# B&R Automation Studio project Hybrid
Automation Studio 6.3.4.31; Oval trak demo with one conveyor segment; technology packages: mappCockpit 6.2.1, mappMotion 6.7.0, mappServices 6.2.0, mappView 6.2.0, OpcUaCs 6.0.0

## Configuration APC2200

CPU 5APC2200.AL14-000, AutomationRuntime 6.3.4, Build 11.3.0, Vc 6.0.0

### Task classes (Cpu.sw)
```
Cyclic#1 (cycle 800 us, tolerance 0 us):
  Main <- Main.prg
DataObjects: McAcpSys
NcDataObjects: McDriveLog
Binaries: FWRules, McAcpSim, ArSvcReg, TCData, McAcpDrv, udbdef, iomap, Config_1, BRRole, arconfig, asfw, Config_5, ashwac, sysconf, User, Config_4, Role, UaCsConfig, ashwd, Config_3, Config_2
Libraries: astime, UaCoal, powerlnk, sys_lib, UaCoalPrv, AsIODiag, runtime, AsBrStr, CoTrace, AsZip, FileIO, MpBase, standard, McBase, McAcpAx, McAxis, MpAxis, McPureVAx, McAcpTrak
```

### Hardware
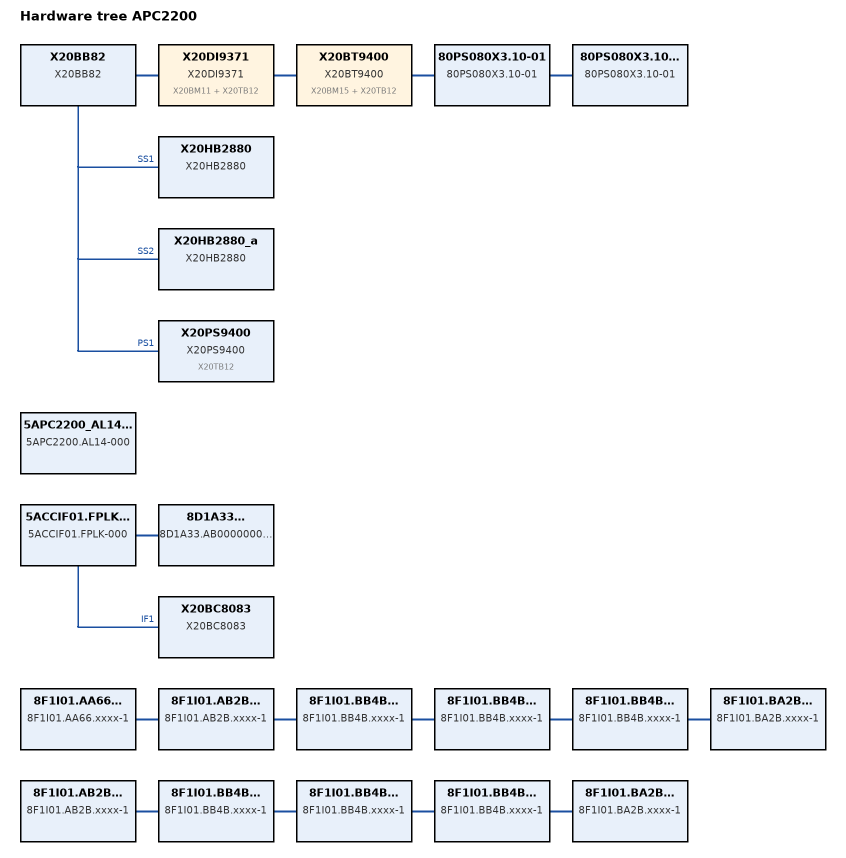
```
5ACCIF01.FPLK-000 : 5ACCIF01.FPLK-000 v1.9.0.0  [PLK2 -> 8D1A33.AB0000000-1.PLK1 [Cable Type=PowerlinkCable, Length=10, Version=1.0.0.3]; SL -> 5APC2200_AL14_000.SL1]
  Connector IF1:
    CycleTime = 800
    EplNatSubnet = 192.168.102.0
    Channel1
    ChannelID1 = McAcpBroadcast
    ChannelType1 = OCTET[120]
5APC2200_AL14_000 : 5APC2200.AL14-000 v2.0.7.0
  Connector IF3:
    AssignedOperatingSystem = ARemb
    ActivateDevice = 1
    HostName = llm-demosystem-ds3
    Mode = Manual
    InternetAddress = 10.43.39.206
    SubnetMask = 255.255.255.0
    InaNodeNumber = 206
    ActivateSnmp = 2
  Connector IF4:
    AssignedOperatingSystem = ARemb
    ActivateDevice = 1
    HostName = llm-demosystem-ds3
    ActivateSnmp = 2
  Connector IF5:
    AssignedOperatingSystem = ARemb
  Connector IF6:
    AssignedOperatingSystem = ARemb
  ConfigurationID = Hybrid_APC910
  Simulation = 1
  MotionLoggerSize = 2048000
  TimerDeviceType = EPLX2X
  TimerDevice = 5ACCIF01.FPLK-000.IF1
  TaskClassIdleTime = 1600
  Cyclic1Duration = 800
  Cyclic1Tolerance = 0
  Cyclic3Duration = 49600
  Cyclic3Tolerance = 49600
  Cyclic8Duration = 9600
  FileDevice1
  FileDeviceName1 = SvgData
  FileDevicePath1 = USER_PATH
  EthernetHostName = llm-demosystem-ds3
  EthernetDefaultGateway = 10.43.39.1
  ActivateFtpServer = 1
  FTPProtocol = 1
  FtpUser1
  FtpUsername1 = Admin
  FtpUserPassword1 = Pdt4iUtP2akYp0fWOPx8iCFOek96otsGjJ7w2jsAU3U=
  FtpUserSalt1 = ubly4TPI
  FTPAccessRight1 = 0
  ActivateWebServer = 1
  WebServerProtocol = 3
  ActivateSdm = 1
80PS080X3.10-01 : 80PS080X3.10-01 v1.7.0.0  [X2X1 -> X20BT9400.X2X1 [Cable Type=X2XCable, Length=10, Version=1.0.0.3]]
  Supervision = off
  ParallelMode01 = on
  VoltageSet01 = 58
  RampMode01 = steep
  ChopperEnable01 = on
80PS080X3.10-01_a : 80PS080X3.10-01 v1.7.0.0  [X2X1 -> 80PS080X3.10-01.X2X2 [Cable Type=X2XCable, Length=10, Version=1.0.0.3]]
  Supervision = off
  ParallelMode01 = on
  VoltageSet01 = 58
  RampMode01 = steep
  ChopperEnable01 = on
8D1A33.AB0000000-1 : 8D1A33.AB0000000-1 v1.0.1.0 (NodeNumber=130)  [PLK1 -> 5ACCIF01.FPLK-000.PLK2 [Cable Type=PowerlinkCable, Length=10, Version=1.0.0.3]]
  DriveConfiguration/Channel[1]/RealAxis:
    AxisReference = gAxis_1
  DriveConfiguration/Channel[1]/RealAxis/MechanicalElements/RotaryToLinearTransformation:
    ReferenceDistance = 0.13
8F1I01.AA66.Seg_0 : 8F1I01.AA66.xxxx-1 v1.0.0.4 (NodeNumber=7)  [PLK1 -> 8F1I01.BA2B.xxxx-1_a.PLK2 [Cable Type=PowerlinkCable, Length=10, Version=1.0.0.3]; PLK2 -> 8F1I01.AB2B.xxxx-1.PLK1 [Cable Type=PowerlinkCable, Length=10, Version=1.0.0.3]; PLK3 -> X20BC8083.PLK2 [Cable Type=PowerlinkCable, Length=10, Version=1.0.0.3]]
  EnableDNA = on
  DriveConfiguration/Segment:
    SegmentReference = Seg_01
8F1I01.AB2B.xxxx-1 : 8F1I01.AB2B.xxxx-1 v1.0.0.4 (NodeNumber=8)  [PLK1 -> 8F1I01.AA66.Seg_0.PLK2 [Cable Type=PowerlinkCable, Length=10, Version=1.0.0.3]; PLK2 -> 8F1I01.BB4B.xxxx-1.PLK1 [Cable Type=PowerlinkCable, Length=10, Version=1.0.0.3]]
  EnableDNA = on
  DriveConfiguration/Segment:
    SegmentReference = Seg_02
8F1I01.AB2B.xxxx-1_a : 8F1I01.AB2B.xxxx-1 v1.0.0.4 (NodeNumber=2)  [PLK2 -> 8F1I01.BB4B.xxxx-1_e.PLK1 [Cable Type=PowerlinkCable, Length=10, Version=1.0.0.3]]
  EnableDNA = on
  DriveConfiguration/Segment:
    SegmentReference = Seg_08
    SegmentSectorReference = SegSec_08
8F1I01.BA2B.xxxx-1 : 8F1I01.BA2B.xxxx-1 v1.0.0.4 (NodeNumber=12)  [PLK1 -> 8F1I01.BB4B.xxxx-1_b.PLK2 [Cable Type=PowerlinkCable, Length=10, Version=1.0.0.3]]
  EnableDNA = on
  DriveConfiguration/Segment:
    SegmentReference = Seg_06
    SegmentSectorReference = SegSec_06
8F1I01.BA2B.xxxx-1_a : 8F1I01.BA2B.xxxx-1 v1.0.0.4 (NodeNumber=6)  [PLK1 -> 8F1I01.BB4B.xxxx-1_c.PLK2 [Cable Type=PowerlinkCable, Length=10, Version=1.0.0.3]; PLK2 -> 8F1I01.AA66.Seg_0.PLK1 [Cable Type=PowerlinkCable, Length=10, Version=1.0.0.3]]
  EnableDNA = on
  DriveConfiguration/Segment:
    SegmentReference = Seg_12
8F1I01.BB4B.xxxx-1 : 8F1I01.BB4B.xxxx-1 v1.0.0.4 (NodeNumber=9)  [PLK1 -> 8F1I01.AB2B.xxxx-1.PLK2 [Cable Type=PowerlinkCable, Length=10, Version=1.0.0.3]; PLK2 -> 8F1I01.BB4B.xxxx-1_a.PLK1 [Cable Type=PowerlinkCable, Length=10, Version=1.0.0.3]]
  EnableDNA = on
  DriveConfiguration/Segment:
    SegmentReference = Seg_03
8F1I01.BB4B.xxxx-1_a : 8F1I01.BB4B.xxxx-1 v1.0.0.4 (NodeNumber=10)  [PLK1 -> 8F1I01.BB4B.xxxx-1.PLK2 [Cable Type=PowerlinkCable, Length=10, Version=1.0.0.3]; PLK2 -> 8F1I01.BB4B.xxxx-1_b.PLK1 [Cable Type=PowerlinkCable, Length=10, Version=1.0.0.3]]
  EnableDNA = on
  DriveConfiguration/Segment:
    SegmentReference = Seg_04
8F1I01.BB4B.xxxx-1_b : 8F1I01.BB4B.xxxx-1 v1.0.0.4 (NodeNumber=11)  [PLK1 -> 8F1I01.BB4B.xxxx-1_a.PLK2 [Cable Type=PowerlinkCable, Length=10, Version=1.0.0.3]; PLK2 -> 8F1I01.BA2B.xxxx-1.PLK1 [Cable Type=PowerlinkCable, Length=10, Version=1.0.0.3]]
  EnableDNA = on
  DriveConfiguration/Segment:
    SegmentReference = Seg_05
8F1I01.BB4B.xxxx-1_c : 8F1I01.BB4B.xxxx-1 v1.0.0.4 (NodeNumber=5)  [PLK1 -> 8F1I01.BB4B.xxxx-1_d.PLK2 [Cable Type=PowerlinkCable, Length=10, Version=1.0.0.3]; PLK2 -> 8F1I01.BA2B.xxxx-1_a.PLK1 [Cable Type=PowerlinkCable, Length=10, Version=1.0.0.3]]
  EnableDNA = on
  DriveConfiguration/Segment:
    SegmentReference = Seg_11
8F1I01.BB4B.xxxx-1_d : 8F1I01.BB4B.xxxx-1 v1.0.0.4 (NodeNumber=4)  [PLK1 -> 8F1I01.BB4B.xxxx-1_e.PLK2 [Cable Type=PowerlinkCable, Length=10, Version=1.0.0.3]; PLK2 -> 8F1I01.BB4B.xxxx-1_c.PLK1 [Cable Type=PowerlinkCable, Length=10, Version=1.0.0.3]]
  EnableDNA = on
  DriveConfiguration/Segment:
    SegmentReference = Seg_10
8F1I01.BB4B.xxxx-1_e : 8F1I01.BB4B.xxxx-1 v1.0.0.4 (NodeNumber=3)  [PLK1 -> 8F1I01.AB2B.xxxx-1_a.PLK2 [Cable Type=PowerlinkCable, Length=10, Version=1.0.0.3]; PLK2 -> 8F1I01.BB4B.xxxx-1_d.PLK1 [Cable Type=PowerlinkCable, Length=10, Version=1.0.0.3]]
  EnableDNA = on
  DriveConfiguration/Segment:
    SegmentReference = Seg_09
    SegmentSectorReference = SegSec_09
X20BB82 : X20BB82 v1.2.0.0
X20BC8083 : X20BC8083 v2.17.0.0 (NodeNumber=129)  [PLK1 -> 5ACCIF01.FPLK-000.IF1 [Cable Type=PowerlinkCable, Length=10, Version=1.0.0.3]; PLK2 -> 8F1I01.AA66.Seg_0.PLK3 [Cable Type=PowerlinkCable, Length=10, Version=1.0.0.3]; SL -> X20BB82.SL1]
  Supervision = off
X20BM11 : X20BM11 v1.1.0.0  [X2X1 -> X20BB82.IF1]
X20BM15 : X20BM15 v1.1.0.0 (NodeNumber=4)  [X2X1 -> X20BM11.X2X2]
X20BT9400 : X20BT9400 v1.3.1.0  [SS1 -> X20TB12_c.SS; SL -> X20BM15.SL1]
  Supervision = off
X20DI9371 : X20DI9371 v1.6.1.0  [SS1 -> X20TB12_a.SS; SL -> X20BM11.SL1]
  Supervision = off
X20HB2880 : X20HB2880 v1.2.1.0  [SS -> X20BB82.SS1]
X20HB2880_a : X20HB2880 v1.2.1.0  [SS -> X20BB82.SS2]
X20PS9400 : X20PS9400 v1.8.1.0  [SS1 -> X20TB12.SS; PS -> X20BB82.PS1]
  Supervision = off
X20TB12 : X20TB12 v1.0.0.0
X20TB12_a : X20TB12 v1.0.0.0
X20TB12_c : X20TB12 v1.0.0.0
```

### Config.mappmotioncfg - 5APC2200_AL14_000/mappMotion/Config.mappmotioncfg
```
Element MappMotionConfiguration (Type=mappmotioncfg)
  Diagnostics:
    Snapshot = Used
      Files:
        FileDevice = SvgData
        Directory = snapshot
        Compression = Not used
        Limits = NotUsed
```

### Config_1.assembly - 5APC2200_AL14_000/mappMotion/Config_1.assembly
```
Element gAssembly_1 (Type=assembly)
  Tracks:
    Track[1]:
      Segments:
        SegmentRef[1] = Seg_01
        SegmentRef[2] = Seg_02
        SegmentRef[3] = Seg_03
        SegmentRef[4] = Seg_04
        SegmentRef[5] = Seg_05
        SegmentRef[6] = Seg_06
        SegmentRef[7] = Seg_07
        SegmentRef[8] = Seg_08
        SegmentRef[9] = Seg_09
        SegmentRef[10] = Seg_10
        SegmentRef[11] = Seg_11
        SegmentRef[12] = Seg_12
      Position:
        SegmentRef = Seg_01
  CommonSegmentSettings:
    ControllerParameters:
      DefaultParameter:
        Controller:
          Position:
            ProportionalGain = 150
          Speed:
            ProportionalGain = 120
          FeedForward:
            TotalMass = 1.25
            ForcePositive = 1
            ForceNegative = 1
        MovementErrorLimits:
          VelocityError = 2.4
    Compensation:
      ElongationCompensation = Active
    ShuttleIdentificationTime = 1
  Shuttles:
    MaxShuttleCount = 20
    ShuttleStereotypes:
      ShuttleStRef[1] = ShuttleStereotype_1
    MagnetPlateConfigurations:
      ShuttleType[1] = 8F1Sx.102.xxxxxx-x
    CollisionAvoidance:
      VirtualShColAvoidanceScope = NoShuttles
    BackupShuttleData = Used
      BackupVar = ::Main:ShuttleData
  AssemblyFeatures:
    AssemblyFeatureRef[1] = AssemblyFeature_Coupling
    AssemblyFeatureRef[2] = AssemblyFeature_Snapshot
    AssemblyFeatureRef[3] = AssemblyFeature_AutoAttach
```

### Config_2.sector - 5APC2200_AL14_000/mappMotion/Config_2.sector
```
Element Sector_1 (Type=sector)
  Type:
    StartSegment:
      SegmentRef = Seg_01
    IntermediateSegments:
      SegmentRef[1] = Seg_02
      SegmentRef[2] = Seg_03
      SegmentRef[3] = Seg_04
      SegmentRef[4] = Seg_05
      SegmentRef[5] = Seg_06
      SegmentRef[6] = Seg_07
      SegmentRef[7] = Seg_08
      SegmentRef[8] = Seg_09
      SegmentRef[9] = Seg_10
      SegmentRef[10] = Seg_11
    EndSegment:
      SegmentRef = Seg_12
      PositionRelativeTo = FromEnd
Element Sector_2 (Type=sector)
  Type:
    StartSegment:
      SegmentRef = Seg_08
    IntermediateSegments:
      SegmentRef[1] = Seg_09
      SegmentRef[2] = Seg_10
      SegmentRef[3] = Seg_11
      SegmentRef[4] = Seg_12
      SegmentRef[5] = Seg_01
      SegmentRef[6] = Seg_02
      SegmentRef[7] = Seg_03
      SegmentRef[8] = Seg_04
      SegmentRef[9] = Seg_05
      SegmentRef[10] = Seg_06
    EndSegment:
      SegmentRef = Seg_07
      PositionRelativeTo = FromEnd
Element Sector_3 (Type=sector)
  Type:
    StartSegment:
      SegmentRef = Seg_01
    EndSegment:
      SegmentRef = Seg_01
      PositionRelativeTo = FromEnd
Element Sector_4 (Type=sector)
  Type:
    StartSegment:
      SegmentRef = Seg_08
    IntermediateSegments:
      SegmentRef[1] = Seg_09
      SegmentRef[2] = Seg_10
      SegmentRef[3] = Seg_11
      SegmentRef[4] = Seg_12
      SegmentRef[5] = Seg_01
      SegmentRef[6] = Seg_02
      SegmentRef[7] = Seg_03
      SegmentRef[8] = Seg_04
      SegmentRef[9] = Seg_05
    EndSegment:
      SegmentRef = Seg_06
      PositionRelativeTo = FromEnd
Element SimSector (Type=sector)
  Type:
    StartSegment:
      SegmentRef = Seg_08
    EndSegment:
      SegmentRef = Seg_08
      Position = 0.07
Element Sector_Check_Free (Type=sector)
  Type = Subsector
    SectorRef = SegSec_06
    Start:
      PositionRelativeTo = FromEnd
    Length = 0.199
```

### Config_3.shuttlestereotype - 5APC2200_AL14_000/mappMotion/Config_3.shuttlestereotype
```
Element ShuttleStereotype_1 (Type=shuttlestereotype)
  MovementLimits:
    Acceleration:
      Acceleration = 30
    Deceleration:
      Deceleration = 30
  JerkFilter = NotUsed
  UserData:
    Size = 12
```

### Config_4.processpoint - 5APC2200_AL14_000/mappMotion/Config_4.processpoint
```
Element ProcessPoint_Entry (Type=processpoint)
  Type:
    SectorRef = SegSec_07
    Position = 0.05
    PositionRelativeTo = FromEnd
    BarrierFunctionality = On
Element ProcessPoint_PreExit (Type=processpoint)
  Type:
    SectorRef = SegSec_06
    Position = 0.2
    PositionRelativeTo = FromEnd
    BarrierFunctionality = On
Element ProcessPoint_Exit (Type=processpoint)
  Type:
    SectorRef = SegSec_06
    Position = 0.135
    PositionRelativeTo = FromEnd
    BarrierFunctionality = On
Element ProcessPoint_Clear (Type=processpoint)
  Type:
    SectorRef = SegSec_09
Element ProcessPoint_AddShuttle (Type=processpoint)
  Type:
    SectorRef = Sector_1
    Position = 0.1
    PositionRelativeTo = FromEnd
    BarrierFunctionality = On
Element ProcessPoint_Safety (Type=processpoint)
  Type:
    SectorRef = SegSec_06
    PositionRelativeTo = FromEnd
    BarrierFunctionality = On
```

### Config_5.virtsegment - 5APC2200_AL14_000/mappMotion/Config_5.virtsegment
```
Element Seg_07 (Type=virtsegment)
  SegmentSectorReference = SegSec_07
```

### Config_6.axis - 5APC2200_AL14_000/mappMotion/Config_6.axis
```
Element gAxis_1 (Type=axis)
  BaseType = Linear
    MeasurementUnit = 5067858
    MeasurementResolution = 0.00001
  MovementLimits:
    Velocity:
      Velocity = 2
    Acceleration:
      Acceleration = 20
    Deceleration:
      Deceleration = 20
```

### Config_7.assemblyfeature - 5APC2200_AL14_000/mappMotion/Config_7.assemblyfeature
```
Element AssemblyFeature_Coupling (Type=assemblyfeature)
  Type:
    CouplingObject[1]:
      Name = Coupling1
      ShuttleCount = 20
Element AssemblyFeature_Snapshot (Type=assemblyfeature)
  Type = AssemblySnapshot
Element AssemblyFeature_AutoAttach (Type=assemblyfeature)
  Type = ShtSectorAutoAttach
    Priority[1]:
      SectorRef = Sector_1
```

## Logical view

Binary libraries used (declarations not repeated): operator, runtime, AsIecCon, astime, AsIODiag, AsBrStr, CoTrace 6.2.1, AsZip, FileIO, MpBase 6.5.0, standard, McBase 6.7.0, McAcpAx 6.7.0, McAxis 6.7.0, MpAxis 6.7.0, McPureVAx 6.7.0, McAcpTrak 6.7.0


### Program Logical/Main (IEC) - Main logic

#### Main.st - Init, cyclic, exit code
```iecst
(*********************************************************************************
 * Copyright: B&R Industrial Automation GmbH
 * Author:    B&R
 * Created:   July 22, 2025/2:17 PM
 * Description: Demo application for an oval trak with one segment as conveyor(hybrid)
 *********************************************************************************)

PROGRAM _INIT

	// Initialize all FUBs once
	MC_BR_AsmPowerOn_0.Assembly			:= ADR(gAssembly_1);
	MC_BR_AsmPowerOff_0.Assembly		:= ADR(gAssembly_1);
	MC_BR_AsmDeleteShuttle_0.Assembly	:= ADR(gAssembly_1);
	MC_BR_AsmDeleteShuttle_0.Command	:= mcACPTRAK_SH_DELETE_ALL;
	MC_BR_AsmReset_0.Assembly			:= ADR(gAssembly_1);
	MC_BR_AsmReadInfo_0.Assembly		:= ADR(gAssembly_1);
	MC_BR_AsmStop_0.Assembly			:= ADR(gAssembly_1);

	MC_BR_SecGetShuttle_0.Sector		:= ADR(Sector_1);

	MC_BR_TrgPointEnable_Entry.ProcessPoint		:= ADR(ProcessPoint_Entry);
	MC_BR_TrgPointReadInfo_Entry.ProcessPoint	:= ADR(ProcessPoint_Entry);

	MC_BR_SegReadInfo_Entry.Segment		:= ADR(Seg_08);
	MC_BR_SegReadInfo_Entry.Enable		:= TRUE;

	MC_BR_TrgPointEnable_Exit.ProcessPoint		:= ADR(ProcessPoint_PreExit);
	MC_BR_TrgPointReadInfo_Exit.ProcessPoint	:= ADR(ProcessPoint_PreExit);

	MC_BR_BarrierCmd_Exit.ProcessPoint			:= ADR(ProcessPoint_PreExit);
	MC_BR_BarrierReadInfo_Exit.ProcessPoint		:= ADR(ProcessPoint_PreExit);
	MC_BR_BarrierReadInfo_Exit.Enable			:= TRUE;

	MC_BR_TrgPointEnable_CheckFree.ProcessPoint	:= ADR(ProcessPoint_Exit);
	MC_BR_SecReadInfo_CheckFree.Sector			:= ADR(Sector_Check_Free);

	MC_BR_TrgPointEnable_Clear.ProcessPoint		:= ADR(ProcessPoint_Clear);
	MC_BR_TrgPointReadInfo_Clear.ProcessPoint	:= ADR(ProcessPoint_Clear);

	MC_BR_SecReadInfo_AddShuttle.Sector	:= ADR(Sector_3);
	MC_BR_SecReadInfo_AddShuttle.Enable	:= TRUE;

	MC_BR_BarrierCmd_AddShuttle.ProcessPoint	:= ADR(ProcessPoint_AddShuttle);

	MC_BR_SecReadInfo_Seg08.Sector		:= ADR(SegSec_08);

	MC_BR_SecReadInfo_SimSector.Sector	:= ADR(SimSector);

	// Initialize axis
	MpAxisBasic_0.MpLink				:= ADR(gAxis_1);
	MpAxisBasic_0.Parameters			:= ADR(AxisParams);
	MpAxisBasic_0.Enable				:= TRUE;

	MpAxisCyclicSet_0.MpLink			:= ADR(gAxis_1);
	MpAxisCyclicSet_0.Parameters		:= ADR(CyclicSetParams);
	MpAxisCyclicSet_0.Enable			:= TRUE;

	// Set the init states
	State		:= INIT;
	StateAxis	:= AXIS_INIT;
	EntryState	:= ENTRY_INIT;
	ExitState	:= EXIT_INIT;
	ClearState	:= CLEAR_INIT;
	AddShuttleState	:= ADDSHUTTLE_INIT;

	// Check if simulation is active
	SimActive	:= DiagCpuIsSimulated();

	// Set default values for the shuttles
	NrOfShuttles	:= 4; // Default number of shuttles for demo application

	// Initialize shuttle positions (spaced evenly) and IDs (ID1, ID2, ID3, ...)
	FOR Index := 0 TO MAX_SHUTTLES_MIN_ONE DO
		ShuttleInitData.Position[Index]	:= DEFAULT_ADD_POSITION + (USINT_TO_LREAL(Index) * SHUTTLE_SPACING);
		brsitoa(Index + 1, ADR(TempIDStr));
		ShuttleInitData.ID[Index] := 'ID';
		brsstrcat(ADR(ShuttleInitData.ID[Index]), ADR(TempIDStr));
	END_FOR;

	AddPosition					:= DEFAULT_ADD_POSITION;
	UserID						:= 'UserID';

	// Set default movement parameter
	Velocity 		:= 2.0;       // m/s - Default trak velocity
	Acceleration 	:= 20.0;      // m/s² - Default acceleration
	Deceleration 	:= 20.0;      // m/s² - Default deceleration
	ConveyorVelocity:= Velocity;

	AutomaticVelocityAdjustment	:= TRUE;

	// Set no error information
	ErrorInfo	:= 'No error';

	ShuttleData;

END_PROGRAM

PROGRAM _CYCLIC

	// Stop the application when the assembly is ready and running
	IF Stop AND (State > GET_SHUTTLE_WAIT OR State = INIT) AND State <> ERROR THEN
		Start	:= FALSE;
		Stop	:= FALSE;
		IF MC_BR_AsmReadInfo_0.AssemblyInfo.PLCopenState = mcACPTRAK_READY THEN
			State	:= STOP_SHUTTLES;
		END_IF;
	END_IF;

	// Reset Halt and Stop when the application is not ready
	// Reset to avoid old flags when starting application
	IF State <> READY THEN
		Halt	:= FALSE;
		Stop	:= FALSE;
	END_IF;

	// Reset the error information
	IF State <> ERROR THEN
		ErrorInfo	:= 'No error';
	END_IF;

	CASE State OF
		// Wait until the start command is set
		// If the application was paused by the Halt command, do not set new shuttles and do not power on again
		INIT:
			MC_BR_AsmReadInfo_0.Enable		:= TRUE;

			// If any virtual shuttles are on the system, get the IDs from end to start and delete all virtual shuttles
			IF MC_BR_AsmReadInfo_0.Valid AND MC_BR_AsmReadInfo_0.AssemblyInfo.ShuttleCount.VirtualShuttles > 0 AND NOT(SimActive) THEN
				State	:= GET_SHUTTLE_IDS_ON_CONVEYOR_INIT;
			END_IF;

			IF Start THEN
				IF Paused AND MC_BR_AsmReadInfo_0.AssemblyInfo.PLCopenState = mcACPTRAK_READY THEN
					State	:= GET_SHUTTLE_INIT;
					Cnt		:= 0;
					UserIDSet	:= TRUE;
				ELSE
					State	:= POWER_ON;
				END_IF;
				MC_BR_AsmReadInfo_0.Enable		:= TRUE;
				MC_BR_SecReadInfo_Seg08.Enable	:= TRUE;
				MC_BR_SecReadInfo_CheckFree.Enable	:= TRUE;
			END_IF;

		// Power on the assembly
		POWER_ON:
			MC_BR_AsmPowerOn_0.Execute		:= TRUE;

			// Close the barrier at the beginning of the conveyor to prevent shuttles to move onto the convoy during cleaning phase
			MC_BR_BarrierCmd_Safety.ProcessPoint	:= ADR(ProcessPoint_Safety);
			MC_BR_BarrierCmd_Safety.Execute			:= TRUE;
			MC_BR_BarrierCmd_Safety.Command			:= mcACPTRAK_BARRIER_CLOSE;

			IF MC_BR_AsmPowerOn_0.Done AND MC_BR_BarrierCmd_Safety.Done THEN
				MC_BR_BarrierCmd_Safety.Execute		:= FALSE;
				MC_BR_AsmPowerOn_0.Execute	:= FALSE;
				Cnt	:= 0;
				UserIDSet	:= FALSE;

				// If the application is simulated, or no shuttles are on the trak, add shuttles to the trak
				IF SimActive AND (NOT(Paused) OR MC_BR_AsmReadInfo_0.AssemblyInfo.ShuttleCount.Count = 0) THEN
					State	:= ADD_SHUTTLES;
					MC_BR_SecAddShuttle_Main.Execute		:= FALSE;
				ELSE
					State	:= GET_SHUTTLE_INIT;
				END_IF;
			ELSIF MC_BR_AsmPowerOn_0.Error THEN
				ErrorInfo	:= 'Error in AsmPowerOn';
				State		:= ERROR;
			END_IF;

		// Add shuttles to the sector
		ADD_SHUTTLES:
			MC_BR_SecAddShuttle_Main.Sector			:= ADR(Sector_1);
			MC_BR_SecAddShuttle_Main.Position		:= ShuttleInitData.Position[Cnt];
			MC_BR_SecAddShuttle_Main.Velocity		:= 0.0;
			MC_BR_SecAddShuttle_Main.AdvancedParameters.UserID	:= ShuttleInitData.ID[Cnt];
			MC_BR_SecAddShuttle_Main.AdvancedParameters.Mode	:= mcACPTRAK_ADD_IMMEDIATE;
			MC_BR_SecAddShuttle_Main.AdvancedParameters.VirtualShuttleID	:= 0;
			MC_BR_SecAddShuttle_Main.AdvancedParameters.MoveCmd				:= mcACPTRAK_MOV_CMD_HALT;
			MC_BR_SecAddShuttle_Main.AdvancedParameters.Velocity			:= 0.0;
			MC_BR_SecAddShuttle_Main.AdvancedParameters.Acceleration		:= 0.0;
			MC_BR_SecAddShuttle_Main.AdvancedParameters.Deceleration		:= 0.0;
			MC_BR_SecAddShuttle_Main.AdvancedParameters.Direction			:= mcDIR_POSITIVE;
			MC_BR_SecAddShuttle_Main.Execute		:= TRUE;

			IF MC_BR_SecAddShuttle_Main.Done THEN
				MC_BR_SecAddShuttle_Main.Execute	:= FALSE;
				Cnt	:= Cnt + 1;

				// When the counter reaches the defined number of shuttles, or no ID is set anymore, get the shuttles
				IF Cnt = NrOfShuttles OR ShuttleInitData.ID[Cnt] = '' THEN
					State	:= GET_SHUTTLE_INIT;
					Cnt		:= 0;
					UserIDSet	:= TRUE;
				END_IF;
			ELSIF MC_BR_SecAddShuttle_Main.Error THEN
				ErrorInfo	:= 'Error in SecAddShuttle';
				State		:= ERROR;
			END_IF;

		// Initialize the SecGetShuttle FUB for non virtual shuttles
		GET_SHUTTLE_INIT:
			NrOfShuttles	:= 0;
			StopConveyor	:= TRUE;
			MC_BR_SecGetShuttle_0.Sector		:= ADR(Sector_1);
			MC_BR_SecGetShuttle_0.Enable		:= TRUE;
			MC_BR_SecGetShuttle_0.Next			:= FALSE;
			MC_BR_SecGetShuttle_0.Mode			:= mcACPTRAK_SEARCH_BACKWARD;
			MC_BR_SecGetShuttle_0.AdvancedParameters.VirtualSelectionMode	:= mcACPTRAK_GET_SH_VIRT_NONVIRTUAL;
			State			:= GET_SHUTTLE_WAIT;

		// Get next shuttle
		GET_SHUTTLE:
			MC_BR_SecGetShuttle_0.Next			:= TRUE;
			State			:= GET_SHUTTLE_WAIT;

		// Get the shuttle
		// When no shuttle remains, move all shuttles
		GET_SHUTTLE_WAIT:
			IF MC_BR_SecGetShuttle_0.Valid THEN
				Shuttle[Cnt]	:= MC_BR_SecGetShuttle_0.Axis;
				Cnt	:= Cnt + 1;

				IF MC_BR_SecGetShuttle_0.RemainingCount = 0 THEN
					MC_BR_SecGetShuttle_0.Enable	:= FALSE;
					MC_BR_SecGetShuttle_0.Next		:= FALSE;
					MC_BR_ElasticMoveVel_0.Execute	:= FALSE;
					NrOfShuttles	:= MC_BR_SecGetShuttle_0.TotalCount;

					// If no shuttle is found or the system runs on a real machine, clean the conveyor
					IF MC_BR_SecGetShuttle_0.TotalCount = 0 AND NOT(SimActive) THEN
						State	:= CLEAN_CONVEYOR;
						Cnt		:= 0;
					// If all UserIDs are set, start the movement
					ELSIF UserIDSet THEN
						State	:= START_MOVEMENT;
						Cnt		:= 0;
					// Set the UserIDs
					ELSE
						State	:= SET_USERID;
					END_IF;
				ELSE
					// If no UserID is set, set the ID
					MC_BR_SecGetShuttle_0.Next		:= FALSE;
					IF UserIDSet THEN
						State	:= GET_SHUTTLE;
					ELSE
						State	:= SET_USERID;
					END_IF;
				END_IF;
			ELSIF MC_BR_SecGetShuttle_0.Error THEN
				ErrorInfo	:= 'Error in SecGetShuttle';
				State		:= ERROR;
			END_IF;

		// Set a UserID to the shuttle
		SET_USERID:
			MC_BR_ShSetUserID_0.Axis	:= ADR(Shuttle[Cnt-1]);
			MC_BR_ShSetUserID_0.UserID	:= ShuttleInitData.ID[Cnt-1];
			MC_BR_ShSetUserID_0.Execute	:= TRUE;

			IF MC_BR_ShSetUserID_0.Done THEN
				MC_BR_ShSetUserID_0.Execute			:= FALSE;
				// If SecGetShuttle is still active, get the next shuttle, otherwise move all shuttles
				IF MC_BR_SecGetShuttle_0.Enable THEN
					State	:= GET_SHUTTLE;
				ELSE
					State	:= START_MOVEMENT;
					Cnt		:= 0;
					UserIDSet	:= TRUE;
				END_IF;
			ELSIF MC_BR_ShSetUserID_0.Error THEN
				ErrorInfo	:= 'Error in ShSetUserID';
				State		:= ERROR;
			END_IF;

		// Move all shuttles
		START_MOVEMENT:
			MC_BR_ElasticMoveVel_0.Axis			:= ADR(Shuttle[Cnt]);
			MC_BR_ElasticMoveVel_0.Velocity		:= Velocity;
			MC_BR_ElasticMoveVel_0.Acceleration	:= Acceleration;
			MC_BR_ElasticMoveVel_0.Deceleration	:= Deceleration;
			MC_BR_ElasticMoveVel_0.Direction	:= mcDIR_POSITIVE;

			// If a shuttle is on the trak and not ready, move the shuttle
			IF StateAxis = AXIS_READY THEN
				MC_BR_ElasticMoveVel_0.Execute	:= TRUE;
			END_IF;

			// Wait for the shuttle to move
			IF EDGEPOS(MC_BR_ElasticMoveVel_0.Active) THEN
				MC_BR_ElasticMoveVel_0.Execute	:= FALSE;
				Cnt	:= Cnt + 1;

				// If all shuttles are moved, go to ready
				IF Cnt = NrOfShuttles THEN
					State	:= READY;
					IF NOT(SimActive) AND NOT(Paused) THEN
						// If the machine was not paused, undetected shuttles can be found on the conveyor
						// Go to the cleaning state
						State	:= CLEAN_CONVEYOR;
						Cnt		:= 0;
					END_IF;
					Paused	:= FALSE;
				END_IF;
			ELSIF MC_BR_ElasticMoveVel_0.Error THEN
				ErrorInfo	:= 'Error in ElasticMoveVel';
				State		:= ERROR;
			END_IF;

		// Clean the conveyor
		// Start the conveyor when the catching is active for a certain amount of time
		// This prevents undetected shuttles on the conveyor
		CLEAN_CONVEYOR:
			IF MC_BR_SecAddShuttle_Clean.Busy THEN
				Paused				:= FALSE;
				StartAxisMovement	:= TRUE;
				StopConveyor		:= FALSE;
			END_IF;

			MC_BR_SecAddShuttle_Clean.Execute	:= TRUE;
			MC_BR_SecAddShuttle_Clean.Sector	:= ADR(Sector_2);
			MC_BR_SecAddShuttle_Clean.Position	:= 0.1;
			MC_BR_SecAddShuttle_Clean.AdvancedParameters.Mode				:= mcACPTRAK_ADD_CATCH;
			MC_BR_SecAddShuttle_Clean.AdvancedParameters.MoveCmd			:= mcACPTRAK_MOV_CMD_ELASTICMOVEVEL;
			MC_BR_SecAddShuttle_Clean.AdvancedParameters.Velocity			:= ConveyorVelocity;
			MC_BR_SecAddShuttle_Clean.AdvancedParameters.Acceleration		:= Acceleration;
			MC_BR_SecAddShuttle_Clean.AdvancedParameters.Deceleration		:= Deceleration;
			MC_BR_SecAddShuttle_Clean.AdvancedParameters.Direction			:= mcDIR_POSITIVE;
			// If no UserID should be recovered take the next from the InitData
			// The IDs are saved when stopping the system
			IF UserIDs[0] = '' THEN
				MC_BR_SecAddShuttle_Clean.AdvancedParameters.UserID			:= ShuttleInitData.ID[NrOfShuttles];
			ELSE
				MC_BR_SecAddShuttle_Clean.AdvancedParameters.UserID			:= UserIDs[Cnt];
			END_IF;

			// Check if a shuttle is catched and increase the number of shuttles on the system
			IF EDGEPOS(MC_BR_SecAddShuttle_Clean.Active) THEN
				MC_BR_SecAddShuttle_Clean.Execute	:= FALSE;

				IF NrOfShuttles < MAX_SHUTTLES THEN
					Shuttle[NrOfShuttles]	:= MC_BR_SecAddShuttle_Clean.Axis;
					NrOfShuttles	:= NrOfShuttles + 1;
					Cnt	:= Cnt + 1;
				ELSE
					ErrorInfo	:= 'Error too many shuttles';
					State		:= ERROR;
				END_IF;
			ELSIF MC_BR_SecAddShuttle_Clean.Error THEN
				ErrorInfo	:= 'Error in SecAddShuttle Catch';
				State		:= ERROR;
			END_IF;

			// Run the conveyor for 1,5s
			Timer.IN	:= TRUE;
			Timer.PT	:= CONVEYOR_CLEAN_TIME; // 1.5 second timeout to detect all shuttles on conveyor

			IF Timer.Q THEN
				Timer.IN	:= FALSE;
				MC_BR_SecAddShuttle_Clean.Execute	:= FALSE;
				State		:= CLEAN_CONVEYOR_ABORT;
			END_IF;

		// Abort the last catch command to free the channel
		CLEAN_CONVEYOR_ABORT:
			MC_BR_SecAddShuttle_Clean.Execute	:= TRUE;
			MC_BR_SecAddShuttle_Clean.AdvancedParameters.Mode				:= mcACPTRAK_ABORT_CATCH;
			IF MC_BR_SecAddShuttle_Clean.Done THEN
				MC_BR_SecAddShuttle_Clean.Execute	:= FALSE;
				// If the system is in errorstop delete all shuttles, otherwise start the process
				IF AbortCleaningCatch THEN
					State	:= DELETE_SHUTTLES;
				ELSE
					State	:= READY;
				END_IF;
				AbortCleaningCatch	:= FALSE;
			ELSIF MC_BR_SecAddShuttle_Clean.Error THEN
				ErrorInfo	:= 'Error in SecAddShuttle Catch Abort';
				State		:= ERROR;
			END_IF;

		// All shuttles added and started
		READY:
			// Open the safety barrier in front of the conveyor
			IF MC_BR_BarrierCmd_Safety.Command = mcACPTRAK_BARRIER_CLOSE THEN
				MC_BR_BarrierCmd_Safety.Execute		:= TRUE;
				MC_BR_BarrierCmd_Safety.Command		:= mcACPTRAK_BARRIER_OPEN;
			END_IF;

			IF MC_BR_BarrierCmd_Safety.Done THEN
				MC_BR_BarrierCmd_Safety.Execute		:= FALSE;
			END_IF;

			StartAxisMovement	:= TRUE;
			StopConveyor		:= FALSE;
			EnableStations		:= TRUE;

			IF Halt THEN
				State			:= HALT_SHUTTLES;
				Paused			:= TRUE;
			END_IF;

		// Stop all shuttles on the assembly after the conveyor stopped --> avoid shuttles from being forgotten on the end of the conveyor
		HALT_SHUTTLES:
			IF MC_BR_AsmReadInfo_0.AssemblyInfo.ShuttleCount.VirtualShuttles = 0 AND MC_BR_AsmReadInfo_0.Valid AND
				MC_BR_SecReadInfo_CheckFree.SectorInfo.InRest AND MC_BR_SecReadInfo_CheckFree.Valid THEN
				StopConveyor	:= TRUE;
				MC_BR_AsmStop_0.Execute	:= TRUE;
			END_IF;

			MC_BR_AsmStop_0.AdvancedParameters.SegmentGroup	:= '';
			MC_BR_AsmStop_0.AdvancedParameters.Deceleration	:= Deceleration;
			IF MC_BR_AsmStop_0.Done THEN
				MC_BR_AsmStop_0.Execute	:= FALSE;
				State		:= INIT;

				FOR Index := 0 TO MAX_SHUTTLES_MIN_ONE DO
					MC_BR_MoveCyclicTcpVel_0[Index].Enable	:= FALSE;
				END_FOR;
			ELSIF MC_BR_AsmStop_0.Error THEN
				ErrorInfo	:= 'Error in AsmStop';
				State		:= ERROR;
			END_IF;

		// Stop all shuttles on the Trak segments
		STOP_SHUTTLES:
			StopConveyor	:= TRUE;
			MC_BR_AsmStop_0.Execute	:= TRUE;
			MC_BR_AsmStop_0.AdvancedParameters.Deceleration	:= Deceleration;
			MC_BR_AsmStop_0.AdvancedParameters.SegmentGroup	:= 'Sector_4';
			IF MC_BR_AsmStop_0.Done THEN
				MC_BR_AsmStop_0.Execute	:= FALSE;
				// If virtual shuttles are on the trak, check the UserIDs to restore at the restart
				IF MC_BR_AsmReadInfo_0.Valid AND MC_BR_AsmReadInfo_0.AssemblyInfo.ShuttleCount.VirtualShuttles > 0 AND NOT(SimActive) THEN
					State	:= GET_SHUTTLE_IDS_ON_CONVEYOR_INIT;
					DeleteAll	:= TRUE;
				ELSE
					State	:= DELETE_SHUTTLES;
				END_IF;
			ELSIF MC_BR_AsmStop_0.Error THEN
				ErrorInfo	:= 'Error in AsmStop';
				State		:= ERROR;
			END_IF;

		// Initialize SecGetShuttle for virtual shuttles
		GET_SHUTTLE_IDS_ON_CONVEYOR_INIT:
			MC_BR_SecGetShuttle_0.Sector		:= ADR(Sector_1);
			MC_BR_SecGetShuttle_0.Enable		:= TRUE;
			MC_BR_SecGetShuttle_0.Next			:= FALSE;
			MC_BR_SecGetShuttle_0.Mode			:= mcACPTRAK_SEARCH_BACKWARD;
			MC_BR_SecGetShuttle_0.AdvancedParameters.VirtualSelectionMode	:= mcACPTRAK_GET_SH_VIRT_VIRTUAL;
			Cnt				:= 0;
			State			:= GET_SHUTTLE_IDS_ON_CONVEYOR_WAIT;

		// Get next virtual shuttle
		GET_SHUTTLE_IDS_ON_CONVEYOR:
			MC_BR_SecGetShuttle_0.Next			:= TRUE;
			State			:= GET_SHUTTLE_IDS_ON_CONVEYOR_WAIT;

		// Get the virtual shuttle
		GET_SHUTTLE_IDS_ON_CONVEYOR_WAIT:
			IF MC_BR_SecGetShuttle_0.Valid THEN
				Shuttle_Conveyor[Cnt]	:= MC_BR_SecGetShuttle_0.Axis;
				Cnt	:= Cnt + 1;

				// When all shuttles are found, read the UserIDs
				IF MC_BR_SecGetShuttle_0.RemainingCount = 0 THEN
					MC_BR_SecGetShuttle_0.Enable	:= FALSE;
					MC_BR_SecGetShuttle_0.Next		:= FALSE;
					NrOfShuttlesOnConveyor	:= MC_BR_SecGetShuttle_0.TotalCount;

					State	:= GET_SHUTTLE_IDS;
					Cnt		:= 0;
				ELSE
					MC_BR_SecGetShuttle_0.Next		:= FALSE;
					State	:= GET_SHUTTLE_IDS_ON_CONVEYOR;
				END_IF;
			ELSIF MC_BR_SecGetShuttle_0.Error THEN
				ErrorInfo	:= 'Error in SecGetShuttle Conveyor';
				State		:= ERROR;
			END_IF;

		// Save all UserIDs in a list
		GET_SHUTTLE_IDS:
			MC_BR_ShReadInfo_GetIDS.Axis	:= ADR(Shuttle_Conveyor[Cnt]);
			MC_BR_ShReadInfo_GetIDS.Enable	:= TRUE;

			IF MC_BR_ShReadInfo_GetIDS.Valid THEN
				MC_BR_ShReadInfo_GetIDS.Enable	:= FALSE;
				UserIDs[Cnt]	:= MC_BR_ShReadInfo_GetIDS.ShuttleInfo.AdditionalInfo.UserID;
				Cnt	:= Cnt + 1;

				// If the application is stopped, delete all shuttles
				IF Cnt >= NrOfShuttlesOnConveyor THEN
					State	:= DELETE_VIRT_SHUTTLES;
				END_IF;
				IF DeleteAll THEN
					DeleteAll:= FALSE;
					State	:= DELETE_SHUTTLES;
				END_IF;
			ELSIF MC_BR_ShReadInfo_GetIDS.Error THEN
				ErrorInfo	:= 'Error in ShReadInfo GetIDs';
				State		:= ERROR;
			END_IF;

		// Delete all shuttles and open the barrier
		DELETE_SHUTTLES:
			UserIDSet		:= FALSE;
			OpenBarrier		:= TRUE;
			EnableStations	:= FALSE;
			CalcShuttle.controlif	:= 0;
			MC_BR_AsmDeleteShuttle_0.Execute	:= TRUE;
			MC_BR_AsmDeleteShuttle_0.Command	:= mcACPTRAK_SH_DELETE_ALL;

			IF MC_BR_AsmDeleteShuttle_0.Done THEN
				MC_BR_AsmDeleteShuttle_0.Execute:= FALSE;
				State		:= POWER_OFF;

				FOR Cnt := 0 TO MAX_SHUTTLES_MIN_ONE DO
					UserIDs[Cnt]	:= '';
				END_FOR;
			ELSIF MC_BR_AsmDeleteShuttle_0.Error THEN
				ErrorInfo	:= 'Error in AsmDeleteShuttle';
				State		:= ERROR;
			END_IF;

		// Delete only virtual shuttles
		DELETE_VIRT_SHUTTLES:
			MC_BR_AsmDeleteShuttle_0.Execute	:= TRUE;
			MC_BR_AsmDeleteShuttle_0.Command	:= mcACPTRAK_SH_DELETE_VIRTUAL;

			IF MC_BR_AsmDeleteShuttle_0.Done THEN
				MC_BR_AsmDeleteShuttle_0.Execute:= FALSE;
				State		:= INIT;
			ELSIF MC_BR_AsmDeleteShuttle_0.Error THEN
				ErrorInfo	:= 'Error in AsmDeleteShuttle Virtual';
				State		:= ERROR;
			END_IF;

		// Power off the assembly
		POWER_OFF:
			StateAxis	:= AXIS_POWER_OFF;
			MC_BR_AsmPowerOff_0.Execute			:= TRUE;

			IF MC_BR_AsmPowerOff_0.Done THEN
				MC_BR_AsmPowerOff_0.Execute		:= FALSE;
				State		:= INIT;
			ELSIF MC_BR_AsmPowerOff_0.Error THEN
				ErrorInfo	:= 'Error in AsmPowerOff';
				State		:= ERROR;
			END_IF;

		// Error state, reset all variables
		ERROR:
			EnableStations	:= FALSE;
			Start			:= FALSE;
			Stop			:= FALSE;
			CalcShuttle.controlif	:= 0;

			MC_BR_AsmPowerOn_0.Execute			:= FALSE;
			MC_BR_AsmPowerOff_0.Execute			:= FALSE;
			MC_BR_AsmDeleteShuttle_0.Execute	:= FALSE;
			MC_BR_AsmReset_0.Execute			:= FALSE;
			MC_BR_AsmReadInfo_0.Enable			:= FALSE;
			MC_BR_AsmStop_0.Execute				:= FALSE;

			MC_BR_SecAddShuttle_Main.Execute	:= FALSE;
			MC_BR_SecAddShuttle_1.Execute		:= FALSE;
			MC_BR_SecGetShuttle_0.Enable		:= FALSE;
			MC_BR_SecReadInfo_Seg08.Enable		:= FALSE;

			MC_BR_SecAddShuttle_Clean.Execute	:= FALSE;
			MC_BR_ShReadInfo_GetIDS.Enable		:= FALSE;
			Timer.IN	:= FALSE;

			MC_BR_ElasticMoveVel_0.Execute		:= FALSE;

			FOR Index := 0 TO MAX_SHUTTLES_MIN_ONE DO
				MC_BR_MoveCyclicTcpVel_0[Index].Enable	:= FALSE;
			END_FOR;

			StopConveyor	:= TRUE;

			// Only set the entry state to error to abort the catch mode
			EntryState		:= ENTRY_ERROR;

	END_CASE;

	CASE StateAxis OF
		// Start the conveyor
		AXIS_INIT:
			IF Start OR (State <> INIT AND State <> POWER_OFF AND State <> DELETE_SHUTTLES AND State <> ERROR) THEN
				StopConveyor:= FALSE;
				StateAxis	:= AXIS_POWER_ON;
			END_IF;

		// Power on the conveyor
		AXIS_POWER_ON:
			IF MpAxisBasic_0.Info.ReadyToPowerOn THEN
				MpAxisBasic_0.Power	:= TRUE;
				IF MpAxisBasic_0.PowerOn THEN
					StateAxis	:= AXIS_HOME;
				END_IF;
			END_IF;

		// Home direct the conveyor
		AXIS_HOME:
			MpAxisBasic_0.Home	:= TRUE;
			IF MpAxisBasic_0.IsHomed THEN
				MpAxisBasic_0.Home	:= FALSE;
				StateAxis		:= AXIS_READY;
			END_IF;

		// Start the cyclic velocity command when no shuttle is on the segment behind the conveyor to avoid a crash
		AXIS_READY:
			IF StartAxisMovement AND (MC_BR_SecReadInfo_Seg08.SectorInfo.ShuttleCount.Count = 0 OR MC_BR_SecReadInfo_Seg08.SectorInfo.ShuttleCount.VirtualShuttles > 0) THEN
				MpAxisCyclicSet_0.MoveCyclicVelocity:= TRUE;
			END_IF;
			IF MC_BR_SegReadInfo_Entry.SegmentInfo.PLCopenState = mcACPTRAK_ERRORSTOP OR StopConveyor THEN
				MpAxisCyclicSet_0.MoveCyclicVelocity:= FALSE;
			END_IF;

		// Power off the conveyor
		AXIS_POWER_OFF:
			MpAxisCyclicSet_0.MoveCyclicVelocity	:= FALSE;
			MpAxisBasic_0.Power	:= FALSE;
			IF MpAxisBasic_0.PowerOn = FALSE THEN
				StateAxis		:= AXIS_INIT;
			END_IF;

		// Error state of the conveyor
		AXIS_ERROR:
			StopConveyor		:= TRUE;
			MpAxisBasic_0.Power	:= FALSE;
			MpAxisBasic_0.Home	:= FALSE;

			MpAxisCyclicSet_0.MoveCyclicVelocity	:= FALSE;

	END_CASE;

	// Check for error in MpAxisBasic
	IF MpAxisBasic_0.Error THEN
		ErrorInfo	:= 'Error in MpAxisBasic';
		StateAxis	:= AXIS_ERROR;
		State		:= ERROR;
	ELSE
		MpAxisBasic_0.ErrorReset	:= FALSE;
	END_IF;

	// Check for error in MpAxisCyclicSet
	IF EDGEPOS(MpAxisCyclicSet_0.Error) THEN
		ErrorInfo	:= 'Error in MpAxisCyclicSet';
		StateAxis	:= AXIS_ERROR;
	ELSE
		MpAxisCyclicSet_0.ErrorReset	:= FALSE;
	END_IF;

	// Check for error in AsmReadInfo
	IF MC_BR_AsmReadInfo_0.Error THEN
		ErrorInfo	:= 'Error in AsmReadInfo';
		State		:= ERROR;
	END_IF;

	// Check for assembly errorstop
	IF MC_BR_AsmReadInfo_0.AssemblyInfo.PLCopenState = mcACPTRAK_ERRORSTOP THEN
		ErrorInfo	:= 'Assembly in errorstop';
		State		:= ERROR;
	END_IF;

	// Check for SecReadInfo error for SegSec_08
	IF MC_BR_SecReadInfo_Seg08.Error THEN
		ErrorInfo	:= 'Error in SecReadInfo Seg08';
		State		:= ERROR;
	END_IF;

	// Check for SecReadInfo error for Sector_Check_Free
	IF MC_BR_SecReadInfo_CheckFree.Error THEN
		ErrorInfo	:= 'Error in SecReadInfo Check_Free';
		State		:= ERROR;
	END_IF;

	// Error reset
	// Do an error reset of the assembly first if assembly and axis are in error
	IF ErrorReset AND (State = ERROR OR StateAxis = AXIS_ERROR) THEN
		IF State = ERROR THEN
			MC_BR_AsmReset_0.Execute		:= TRUE;

			IF MC_BR_AsmReset_0.Done THEN
				IF StateAxis <> AXIS_ERROR THEN
					ErrorReset	:= FALSE;
					ErrorInfo	:= 'No error';
				END_IF;
				MC_BR_AsmReset_0.Execute	:= FALSE;
				State		:= INIT;
				OpenBarrier	:= TRUE;

				// If the catch is active for cleaning the conveyor, abort the catch
				IF MC_BR_SecAddShuttle_Clean.Active THEN
					State	:= CLEAN_CONVEYOR_ABORT;
					AbortCleaningCatch	:= TRUE;
				END_IF;

				// No shuttle will be catched after poweron the conveyor
				// Therefore all shuttles will be deleted in the simulation to restart the application
				IF SimActive THEN
					State	:= DELETE_SHUTTLES;
				END_IF;
			ELSIF MC_BR_AsmReset_0.Error THEN
				MC_BR_AsmReset_0.Execute	:= FALSE;
				ErrorInfo	:= 'Error in AsmReset';
				State		:= ERROR;
			END_IF;
		END_IF;

		IF StateAxis = AXIS_ERROR THEN
			StateAxis	:= AXIS_POWER_OFF;
			MpAxisBasic_0.ErrorReset	:= TRUE;
			MpAxisCyclicSet_0.ErrorReset:= TRUE;
			ErrorReset	:= FALSE;
			ErrorInfo	:= 'No error';
		END_IF;
	END_IF;

	// Station actions
	EntrySegment;
	ExitSegment;
	Clear;
	AddNewShuttle;
	CalcAutomaticVelocity;

	// Add messages, timestamps and image index to the list
	IF AddMessage THEN
		AddMessage	:= FALSE;
		FOR Index := 19 TO 1 BY -1 DO
			Messages[Index]		:= Messages[Index-1];
			ImageIndex[Index]	:= ImageIndex[Index-1];
			Timestamps[Index]	:= Timestamps[Index-1];
		END_FOR;
		Messages[0]		:= Message;
		ImageIndex[0]	:= AddImage;
		DTGetTime_0.enable	:= TRUE;
	END_IF;

	DTGetTime_0();

	IF DTGetTime_0.status = 0 THEN
		DTGetTime_0.enable	:= FALSE;
		Timestamps[0]		:= DTGetTime_0.DT1;
	END_IF;

	// Reset the start command after all states are run through
	Start		:= FALSE;

	// Call all FUBs
	MC_BR_AsmPowerOn_0();
	MC_BR_AsmPowerOff_0();
	MC_BR_AsmDeleteShuttle_0();
	MC_BR_AsmReset_0();
	MC_BR_AsmReadInfo_0();
	MC_BR_AsmStop_0();

	MC_BR_SecAddShuttle_Main();
	MC_BR_SecAddShuttle_0();
	MC_BR_SecAddShuttle_1();
	MC_BR_SecAddShuttle_Clean();
	MC_BR_SecGetShuttle_0();
	MC_BR_SecReadInfo_Seg08();
	MC_BR_SecReadInfo_CheckFree();

	MC_BR_ShSetUserID_0();

	MC_BR_ElasticMoveVel_0();

	MC_BR_BarrierCmd_Safety();

	Timer();

	MC_BR_ShReadInfo_GetIDS();

	MpAxisBasic_0();

	MpAxisCyclicSet_0.CyclicVelocity	:= ConveyorVelocity;
	MpAxisCyclicSet_0();

	FOR Index := 0 TO MAX_SHUTTLES_MIN_ONE DO
		// Read shuttle information if available
		IF Shuttle[Index].controlif <> 0 AND State > SET_USERID AND State < DELETE_SHUTTLES AND Index < NrOfShuttles THEN
			MC_BR_ShReadInfo_Main[Index].Axis	:= ADR(Shuttle[Index]);
			MC_BR_ShReadInfo_Main[Index].Enable	:= TRUE;
		ELSE
			MC_BR_ShReadInfo_Main[Index].Enable	:= FALSE;
		END_IF;
		MC_BR_ShReadInfo_Main[Index]();

		IF MC_BR_ShReadInfo_Main[Index].ShuttleInfo.AdditionalInfo.PLCopenState = mcAXIS_ERRORSTOP THEN
			ErrorInfo	:= 'Errorstop in Shuttle';
			State		:= ERROR;
		ELSIF MC_BR_ShReadInfo_Main[Index].Error THEN
			ErrorInfo	:= 'Error in ShReadInfo';
			State		:= ERROR;
		END_IF;

		// Reset MoveCyclicTcpVel after another command took over the shuttle
		MC_BR_MoveCyclicTcpVel_0[Index].Axis			:= ADR(Shuttle[Index]);
		MC_BR_MoveCyclicTcpVel_0[Index].CyclicVelocity	:= MpAxisBasic_0.Velocity;

		IF MC_BR_MoveCyclicTcpVel_0[Index].CommandAborted THEN
			MC_BR_MoveCyclicTcpVel_0[Index].Enable		:= FALSE;
		END_IF;

		MC_BR_MoveCyclicTcpVel_0[Index]();
		IF MC_BR_MoveCyclicTcpVel_0[Index].Error THEN
			ErrorInfo	:= 'Error in MoveCyclicTcpVel';
			State		:= ERROR;
		END_IF;
	END_FOR;

	// Track state changes for debugging
	IF State <> LastState THEN
		// Shift history
		FOR Index := 9 TO 1 BY -1 DO
			StateHistory[Index] := StateHistory[Index-1];
		END_FOR;
		StateHistory[0] := LastState;
		LastState := State;
	END_IF;

	AutomaticVelocityAdjNotActive	:= NOT(AutomaticVelocityAdjustment);

	MachineRunning	:= State = INIT;

END_PROGRAM

PROGRAM _EXIT

	MpAxisBasic_0.Enable		:= FALSE;
	MpAxisBasic_0();

	MpAxisCyclicSet_0.Enable	:= FALSE;
	MpAxisCyclicSet_0();

END_PROGRAM
```

#### Types.typ - Local data types
```iecst
TYPE
	StateEnum :
		( (*Main state enum*)
		INIT, (*Initial state*)
		POWER_ON, (*Power on the assembly*)
		ADD_SHUTTLES, (*Add shuttles to the sector*)
		GET_SHUTTLE_INIT, (*Get shuttles on the assembly - init FUBs*)
		GET_SHUTTLE, (*Get shuttle on the assembly*)
		GET_SHUTTLE_WAIT, (*Wait for shuttle to be read*)
		SET_USERID, (*Set a UserID to the shuttle*)
		START_MOVEMENT, (*Start movement for all shuttles and axis*)
		CLEAN_CONVEYOR, (*Clean the conveyor from missing shuttles*)
		CLEAN_CONVEYOR_ABORT, (*Abort the catch from the cleaning state*)
		READY, (*Application running*)
		HALT_SHUTTLES, (*Execute a stop without power off and deletion of shuttles*)
		STOP_SHUTTLES, (*Stop all shuttles from the Stop command*)
		DELETE_SHUTTLES, (*Delete all shuttles*)
		DELETE_VIRT_SHUTTLES, (*Delete only virtual shuttles*)
		GET_SHUTTLE_IDS_ON_CONVEYOR_INIT, (*Initialize SecGetShuttle to catch all virtual shuttles on the system*)
		GET_SHUTTLE_IDS_ON_CONVEYOR, (*Get the next shuttle*)
		GET_SHUTTLE_IDS_ON_CONVEYOR_WAIT, (*If a shuttle is found, get the reference until all shuttles found*)
		GET_SHUTTLE_IDS, (*Iterate through the list of found shuttles and get the UserIDs*)
		POWER_OFF, (*Power off the assembly*)
		ERROR (*Error*)
		);
	StateAxisEnum :
		( (*Axis state enum*)
		AXIS_INIT, (*Initial state*)
		AXIS_POWER_ON, (*Power on the axis*)
		AXIS_HOME, (*Home the axis*)
		AXIS_READY, (*Axis is ready and can be used*)
		AXIS_POWER_OFF, (*Power off the axis*)
		AXIS_ERROR (*Error*)
		);
	EntryStateEnum :
		( (*Entry state enum*)
		ENTRY_INIT, (*Initial state*)
		ENTRY_CHECK_TRIGGER, (*Check if shuttle moved over the trigger*)
		ENTRY_GET_SHUTTLE, (*Get the shuttle reference from the trigger*)
		ENTRY_GET_SHUTTLEID, (*Get the shuttle ID to catch the virtual shuttle*)
		ENTRY_CATCH_SHUTTLE, (*Catch the shuttles*)
		ENTRY_ERROR, (*Error*)
		ENTRY_ABORT_CATCH (*Abort the catch mode*)
		);
	ExitStateEnum :
		( (*Exit state enum*)
		EXIT_INIT, (*Initial state*)
		EXIT_CHECK_TRIGGER, (*Check if shuttle moved over the trigger*)
		EXIT_GET_SHUTTLE, (*Get the shuttle reference from the trigger*)
		EXIT_GET_SHUTTLEID, (*Get the shuttle ID to catch the virtual shuttle*)
		EXIT_CYCMOVEVEL, (*Execute cyclic velocity*)
		EXIT_ERROR (*Error*)
		);
	ClearStateEnum :
		( (*Clear state enum*)
		CLEAR_INIT, (*Initial state*)
		CLEAR_CHECK_TRIGGER, (*Check if shuttle moved over the trigger*)
		CLEAR_GET_SHUTTLE, (*Get the shuttle reference from the trigger*)
		CLEAR_MOVE_SH_ELASTIC, (*Move the shuttle elastic*)
		CLEAR_ERROR (*Error*)
		);
	AddShuttleStateEnum :
		( (*Add shuttles to the trak enum*)
		ADDSHUTTLE_INIT, (*Initial state*)
		ADDSHUTTLE_CLOSE_BARRIER, (*Close the barrier*)
		ADDSHUTTLE_ADD_SHUTTLE, (*Add shuttle to the trak*)
		ADDSHUTTLE_CHECK_CREATED, (*Check if the shuttle was created*)
		ADDSHUTTLE_POWER_OFF_SEGMENT,
		ADDSHUTTLE_POWER_ON_SEGMENT,
		ADDSHUTTLE_GET_SHUTTLE,
		ADDSHUTTLE_SET_USERID,
		ADDSHUTTLE_MOVESHUTTLE,
		ADDSHUTTLE_OPEN_BARRIER, (*Open the barrier*)
		ADDSHUTTLE_RESET, (*Reset all FUBs*)
		ADDSHUTTLE_ERROR (*Error*)
		);
	ShuttleInitDataType : 	STRUCT  (*Initial data for creating shuttles*)
		Position : ARRAY[0..MAX_SHUTTLES_MIN_ONE]OF LREAL; (*Position on the sector*)
		ID : ARRAY[0..MAX_SHUTTLES_MIN_ONE]OF STRING[32]; (*ID of the shuttle*)
	END_STRUCT;
END_TYPE
```

#### Variables.var - Local variables
```iecst
(**********************************************************************************************************************************************************************************************************************)
VAR CONSTANT
	MAX_SHUTTLES : USINT := 20; (*Max shuttles on the trak*)
	MAX_SHUTTLES_MIN_ONE : USINT := MAX_SHUTTLES-1; (*Max shuttles on the trak minus one*)
	CONVEYOR_CLEAN_TIME : TIME := T#1500ms; (*Time to run the conveyor during cleaning phase*)
	DEFAULT_ADD_POSITION : REAL := 0.1; (*Default position for adding shuttles*)
	ENTRY_POSITION_THRESHOLD : REAL := 0.0; (*Position threshold for entry segment*)
	CLEAR_POSITION_THRESHOLD : REAL := 0.2; (*Position threshold for velocity adjustment calculation*)
	SHUTTLE_SPACING : LREAL := 0.1; (*Spacing between shuttles during initialization*)
END_VAR
(**********************************************************************************************************************************************************************************************************************)
VAR
	MC_BR_AsmPowerOn_0 : MC_BR_AsmPowerOn_AcpTrak; (*FUB to power on the assembly*)
	MC_BR_AsmPowerOff_0 : MC_BR_AsmPowerOff_AcpTrak; (*FUB to power off the assembly*)
	MC_BR_AsmDeleteShuttle_0 : MC_BR_AsmDeleteShuttle_AcpTrak; (*FUB to delete shuttles*)
	MC_BR_AsmReset_0 : MC_BR_AsmReset_AcpTrak; (*FUB to reset the assembly errors*)
	MC_BR_AsmStop_0 : MC_BR_AsmStop_AcpTrak; (*FUB to stop all shuttles on the assembly*)
	MC_BR_AsmReadInfo_0 : MC_BR_AsmReadInfo_AcpTrak; (*FUB to read assembly information*)
	MC_BR_SecAddShuttle_Main : MC_BR_SecAddShuttle_AcpTrak; (*FUB to add shuttles to the sector*)
	MC_BR_SecGetShuttle_0 : MC_BR_SecGetShuttle_AcpTrak; (*FUB to read all shuttle references*)
	MC_BR_ShSetUserID_0 : MC_BR_ShSetUserID_AcpTrak; (*FUB to set the UserID*)
	MC_BR_SecAddShuttle_Clean : MC_BR_SecAddShuttle_AcpTrak; (*FUB to catch all shuttles during the cleaning phase of the conveyor*)
	MC_BR_SecReadInfo_Seg08 : MC_BR_SecReadInfo_AcpTrak; (*FUB to read the sector info for SegSec_08*)
	MC_BR_ElasticMoveVel_0 : MC_BR_ElasticMoveVel_AcpTrak; (*FUB to move all shuttles elastic*)
	MC_BR_ShReadInfo_Main : ARRAY[0..MAX_SHUTTLES_MIN_ONE] OF MC_BR_ShReadInfo_AcpTrak; (*FUB to read the shuttle info*)
	MC_BR_BarrierCmd_Safety : MC_BR_BarrierCommand_AcpTrak; (*FUB to control the barrier at the beginning of the conveyor*)
	MpAxisBasic_0 : MpAxisBasic; (*FUB to use a single axis*)
	AxisParams : MpAxisBasicParType; (*Parameter structure for MpAxisBasic*)
	MpAxisCyclicSet_0 : MpAxisCyclicSet; (*FUB to override cyclically values of the axis (velocity)*)
	CyclicSetParams : MpAxisCyclicSetParType; (*Parameter structure for MpAxisCyclicSet*)
	MC_BR_MoveCyclicTcpVel_0 : ARRAY[0..MAX_SHUTTLES_MIN_ONE] OF MC_BR_MoveCyclicTcpVel_AcpTrak; (*FUB to move shuttles cyclic velocity*)
	Timer : TON; (*Time to wait to clean the conveyor from shuttles*)
	AbortCleaningCatch : BOOL; (*If an error occurs catching shuttles during the cleaning phase, abort the catch and not go to READY*)
END_VAR
(**********************************************************************************************************************************************************************************************************************)
VAR
	State : StateEnum; (*Main state*)
	ErrorInfo : STRING[80]; (*Error information*)
	SimActive : BOOL; (*Simulation active flag*)
	StateAxis : StateAxisEnum; (*Axis state*)
	Start : BOOL; (*Start command*)
	Stop : BOOL; (*Stop command*)
	Halt : BOOL; (*Halt command*)
	AutomaticVelocityAdjustment : BOOL; (*Automatic velocity adjustment mode*)
	AutomaticVelocityAdjNotActive : BOOL; (*Automatic velocity adjustment not active --> mappView*)
	ErrorReset : BOOL; (*Error reset command*)
	ConveyorVelocity : REAL; (*Cyclic velocity for the conveyor and shuttles on the conveyor*)
	Shuttle : ARRAY[0..MAX_SHUTTLES_MIN_ONE] OF McAxisType; (*Shuttle objects*)
	ShuttleInitData : ShuttleInitDataType; (*Initial shuttle data, Position, ID*)
	TempIDStr : STRING[20]; (*Temporary string for ID conversion*)
	NrOfShuttles : UINT; (*Number of shuttles on the system*)
	Velocity : REAL; (*Global velocity for the trak*)
	Acceleration : REAL; (*Global acceleration*)
	Deceleration : REAL; (*Global deceleration*)
	EnableStations : BOOL; (*All stations are enabled*)
	StartAxisMovement : BOOL; (*Start the cyclic movement of the axis*)
	StopConveyor : BOOL; (*Flag to stop the conveyor*)
	Paused : BOOL; (*Paused flag*)
	UserIDSet : BOOL; (*Flag to check if UserID is already set*)
	Cnt : USINT; (*Counter*)
	UserIDs : ARRAY[0..MAX_SHUTTLES_MIN_ONE] OF STRING[80]; (*UserIDs of the Shuttles*)
	ShuttleData : ARRAY[0..1599] OF USINT; (*DataBuffer to recover UserData depending on the UserID*)
	DeleteAll : BOOL; (*If the whole application is stopped delete all shuttles (not only the virtual shuttles)*)
	MachineRunning : BOOL; (*Bool for mappView Visu if machine is running*)
END_VAR
(**********************************************************************************************************************************************************************************************************************)
VAR
	MC_BR_ShReadInfo_GetIDS : MC_BR_ShReadInfo_AcpTrak; (*FUB to read the Shuttle UserID when stopping/errorstop the application*)
	Shuttle_Conveyor : ARRAY[0..MAX_SHUTTLES_MIN_ONE] OF McAxisType; (*Virtual shuttles found while reading the UserIDs of the virtual shuttles*)
	NrOfShuttlesOnConveyor : UINT; (*Number of virtual shuttles on the conveyor, check how many shuttle UserIDs need to be found*)
END_VAR
(**********************************************************************************************************************************************************************************************************************)
VAR
	EntryState : EntryStateEnum; (*Entry state (Exit conveyor)*)
	EntryShuttle : McAxisType; (*Shuttle entered the trak*)
	VirtShID : UDINT; (*Virtual shuttle ID of the entered shuttle*)
	MC_BR_TrgPointEnable_Entry : MC_BR_TrgPointEnable_AcpTrak; (*FUB to get Trigger events*)
	MC_BR_TrgPointReadInfo_Entry : MC_BR_TrgPointReadInfo_AcpTrak; (*FUB to read shuttle from trigger event*)
	MC_BR_ShReadInfo_Entry : MC_BR_ShReadInfo_AcpTrak; (*FUB to read shuttle information*)
	MC_BR_SegReadInfo_Entry : MC_BR_SegReadInfo_AcpTrak; (*FUB to read segment information*)
	MC_BR_SecReadInfo_SimSector : MC_BR_SecReadInfo_AcpTrak; (*FUB to read sector information*)
	MC_BR_SecAddShuttle_0 : MC_BR_SecAddShuttle_AcpTrak; (*FUB to catch shuttle*)
	MC_BR_SecAddShuttle_1 : MC_BR_SecAddShuttle_AcpTrak; (*FUB to catch shuttle*)
END_VAR
(**********************************************************************************************************************************************************************************************************************)
VAR
	ExitState : ExitStateEnum; (*Exit state (Entry conveyor)*)
	ExitShuttle : McAxisType; (*Shuttle exit the trak*)
	AddTicket : BOOL; (*Add ticket to the barrier*)
	MC_BR_TrgPointEnable_Exit : MC_BR_TrgPointEnable_AcpTrak; (*FUB to get Trigger events*)
	MC_BR_TrgPointReadInfo_Exit : MC_BR_TrgPointReadInfo_AcpTrak; (*FUB to read shuttle from trigger event*)
	MC_BR_ShReadInfo_Exit : MC_BR_ShReadInfo_AcpTrak; (*FUB to read shuttle information*)
	MC_BR_BarrierCmd_Exit : MC_BR_BarrierCommand_AcpTrak; (*FUB to control the barrier*)
	MC_BR_BarrierReadInfo_Exit : MC_BR_BarrierReadInfo_AcpTrak; (*FUB to read the barrier information*)
	MC_BR_SecReadInfo_CheckFree : MC_BR_SecReadInfo_AcpTrak; (*FUB to check if the segment behind the barrier is free*)
	MC_BR_TrgPointEnable_CheckFree : MC_BR_TrgPointEnable_AcpTrak; (*FUB to get Trigger events if shuttle distance is high enough*)
END_VAR
(**********************************************************************************************************************************************************************************************************************)
VAR
	ClearState : ClearStateEnum; (*Clear state*)
	ClearShuttle : McAxisType; (*Shuttle at the clear station*)
	MC_BR_TrgPointEnable_Clear : MC_BR_TrgPointEnable_AcpTrak; (*FUB to get Trigger events*)
	MC_BR_TrgPointReadInfo_Clear : MC_BR_TrgPointReadInfo_AcpTrak; (*FUB to read shuttle from trigger event*)
	MC_BR_ElasticMoveVel_Clear : MC_BR_ElasticMoveVel_AcpTrak; (*FUB to move elastic velocity*)
	Index : USINT; (*Index counter variable*)
END_VAR
(**********************************************************************************************************************************************************************************************************************)
VAR
	Message : STRING[80]; (*Message to add to the list*)
	Messages : ARRAY[0..19] OF STRING[80]; (*Messages for the visu*)
	ImageIndex : ARRAY[0..19] OF USINT; (*Image index for the visu*)
	AddMessage : BOOL; (*Add the new message to the list*)
	AddImage : USINT; (*Add the new image to the list*)
	Timestamps : ARRAY[0..19] OF DATE_AND_TIME; (*List with timestamps for the visu*)
	DTGetTime_0 : DTGetTime; (*FUB to read the timestamp*)
END_VAR
(**********************************************************************************************************************************************************************************************************************)
VAR
	AddShuttleState : AddShuttleStateEnum; (*State enum for adding the shuttle*)
	AddShuttle : BOOL; (*Add a shuttle to the trak*)
	OpenBarrier : BOOL; (*Open the barrier*)
	AddPosition : LREAL; (*Position where the shuttle should be added*)
	ConfirmShuttleAdded : BOOL; (*On the PLC, confirm that the shuttles are placed on the assembly*)
	UserID : STRING[32]; (*UserID of the added shuttle*)
	MC_BR_SecAddShuttle_AddShuttle : MC_BR_SecAddShuttle_AcpTrak; (*FUB to add a shuttle*)
	MC_BR_SecReadInfo_AddShuttle : MC_BR_SecReadInfo_AcpTrak; (*FUB to read sector info*)
	MC_BR_BarrierCmd_AddShuttle : MC_BR_BarrierCommand_AcpTrak; (*FUB to control the barrier*)
	MC_BR_SegPowerOff_AddShuttle : MC_BR_SegPowerOff_AcpTrak; (*FUB to power off the segment*)
	MC_BR_SegPowerOn_AddShuttle : MC_BR_SegPowerOn_AcpTrak; (*FUB to power on the segment*)
	MC_BR_SecGetShuttle_AddShuttle : MC_BR_SecGetShuttle_AcpTrak; (*FUB to read the shuttles on the sector*)
	MC_BR_ShSetUserID_AddShuttle : MC_BR_ShSetUserID_AcpTrak; (*FUB to set the UserID*)
	MC_BR_ElasticMoveVel_AddShuttle : MC_BR_ElasticMoveVel_AcpTrak; (*FUB to move the shuttle*)
	AddedShuttle : McAxisType; (*Shuttle reference that is read*)
	BarrierClosed_AddShuttle : BOOL; (*Barrier closed, used for mappView to enable confirm button*)
	AxisOld : McAxisType; (*Temp variable to check controlif changed*)
END_VAR
(**********************************************************************************************************************************************************************************************************************)
VAR
	MC_BR_ShReadInfo_Calc : MC_BR_ShReadInfo_AcpTrak; (*FUB to read the shuttle info*)
	CalcShuttle : McAxisType; (*Shuttle reference of the last catched shuttle*)
	OldShuttle_Calc : McAxisType; (*Old shuttle reference to check if new one is available*)
END_VAR
(**********************************************************************************************************************************************************************************************************************)
VAR
	LastState : StateEnum; (*Last main state for change tracking*)
	StateHistory : ARRAY[0..9] OF StateEnum; (*History of last 10 states for debugging*)
END_VAR
```

#### EntrySegment.st - Entry to the trak from the conveyor
```iecst
(*********************************************************************************
 * Copyright: B&R Industrial Automation GmbH
 * Author:    B&R
 * Created:   July 22, 2025/2:18 PM
 * Description: Entry to the trak from the conveyor, catch all shuttles
 *********************************************************************************)

ACTION EntrySegment:

	// Reset the state machine and all FUBs after a stop command
	IF EnableStations = FALSE AND EntryState <> ENTRY_INIT AND EntryState <> ENTRY_ABORT_CATCH THEN
		EntryState	:= ENTRY_ERROR;
	END_IF;

	CASE EntryState OF
		// Wait for enabling the station
		ENTRY_INIT:
			IF EnableStations AND NOT(Paused) THEN
				EntryState	:= ENTRY_CHECK_TRIGGER;
			END_IF;

			IF MC_BR_SecAddShuttle_0.Active OR MC_BR_SecAddShuttle_1.Active THEN
				EntryState	:= ENTRY_ABORT_CATCH;
			END_IF;

		// Check for shuttle passed the trigger
		ENTRY_CHECK_TRIGGER:
			MC_BR_TrgPointEnable_Entry.Enable		:= TRUE;
			MC_BR_ShReadInfo_Entry.Enable			:= FALSE;
			MC_BR_SecReadInfo_SimSector.Enable		:= TRUE;

			IF MC_BR_TrgPointEnable_Entry.Valid AND MC_BR_TrgPointEnable_Entry.EventCount > 0 THEN
				EntryState	:= ENTRY_GET_SHUTTLE;
			ELSIF MC_BR_TrgPointEnable_Entry.Error THEN
				ErrorInfo	:= 'Error in TrgPointEnable Entry';
				State		:= ERROR;
				EntryState	:= ENTRY_ERROR;
			END_IF;

		// Get the passing shuttle
		ENTRY_GET_SHUTTLE:
			MC_BR_TrgPointReadInfo_Entry.Execute	:= TRUE;

			IF MC_BR_TrgPointReadInfo_Entry.Done THEN
				MC_BR_TrgPointReadInfo_Entry.Execute	:= FALSE;
				EntryShuttle	:= MC_BR_TrgPointReadInfo_Entry.TrgPointInfo.Axis;
				EntryState		:= ENTRY_GET_SHUTTLEID;
			ELSIF MC_BR_TrgPointReadInfo_Entry.Error THEN
				ErrorInfo	:= 'Error in TrgPointReadInfo Entry';
				State		:= ERROR;
				EntryState	:= ENTRY_ERROR;
			END_IF;

		// Get the shuttle virtual ID and velocity (for sim)
		ENTRY_GET_SHUTTLEID:
			MC_BR_ShReadInfo_Entry.Axis		:= ADR(EntryShuttle);
			MC_BR_ShReadInfo_Entry.Enable	:= TRUE;

			IF MC_BR_ShReadInfo_Entry.Valid THEN
				VirtShID	:= MC_BR_ShReadInfo_Entry.ShuttleInfo.AdditionalInfo.ID;
				EntryState	:= ENTRY_CATCH_SHUTTLE; // Virtual ID retrieved, ready to catch real shuttle

				Message		:= 'Shuttle "';
				brsstrcat(ADR(Message),ADR(MC_BR_ShReadInfo_Entry.ShuttleInfo.AdditionalInfo.UserID));
				brsstrcat(ADR(Message),ADR('" left the conveyor and entered the trak'));
				AddMessage	:= TRUE;  // Queue status message for visualization
				AddImage	:= 0;       // Icon index 0: Shuttle entering trak
			ELSIF MC_BR_ShReadInfo_Entry.Error THEN
				ErrorInfo	:= 'Error in ShReadInfo Entry';
				State		:= ERROR;
				EntryState	:= ENTRY_ERROR;
			END_IF;

		// Catch the shuttle
		// Use two FUBs to be able to catch two shuttles if one is waiting
		ENTRY_CATCH_SHUTTLE:
			IF NOT(MC_BR_SecAddShuttle_0.Execute) THEN
				// Set velocity if the simulation is active
				// If the simulation is active, wait until the shuttle reached the position before catching the shuttle
				IF SimActive AND MC_BR_ShReadInfo_Entry.ShuttleInfo.CurrentValues.SegmentPosition.Position >= ENTRY_POSITION_THRESHOLD AND MC_BR_ShReadInfo_Entry.ShuttleInfo.CurrentValues.SegmentPosition.Segment.controlif = Seg_08.controlif (*AND MC_BR_SecReadInfo_SimSector.SectorInfo.ShuttleCount.Count = 0 AND MC_BR_SecReadInfo_SimSector.Valid*) THEN
					MC_BR_SecAddShuttle_0.Velocity	:= ConveyorVelocity;
					MC_BR_SecAddShuttle_0.Execute	:= TRUE;
					EntryState	:= ENTRY_CHECK_TRIGGER;
				ELSIF NOT(SimActive) THEN
					MC_BR_SecAddShuttle_0.Execute	:= TRUE;
					EntryState	:= ENTRY_CHECK_TRIGGER;
				END_IF;
				MC_BR_SecAddShuttle_0.Sector	:= ADR(Sector_2);
				MC_BR_SecAddShuttle_0.Position	:= 0.0;
				MC_BR_SecAddShuttle_0.AdvancedParameters.Mode				:= mcACPTRAK_ADD_CATCH; // Catch mode: convert virtual to real shuttle
				MC_BR_SecAddShuttle_0.AdvancedParameters.VirtualShuttleID	:= VirtShID; // Link to virtual shuttle on conveyor
				MC_BR_SecAddShuttle_0.AdvancedParameters.MoveCmd			:= mcACPTRAK_MOV_CMD_ELASTICMOVEVEL; // Continue with elastic movement
				MC_BR_SecAddShuttle_0.AdvancedParameters.Velocity			:= ConveyorVelocity;
				MC_BR_SecAddShuttle_0.AdvancedParameters.Acceleration		:= Acceleration;
				MC_BR_SecAddShuttle_0.AdvancedParameters.Deceleration		:= Deceleration;
				MC_BR_SecAddShuttle_0.AdvancedParameters.Direction			:= mcDIR_POSITIVE;
				MC_BR_SecAddShuttle_0.AdvancedParameters.UserID				:= '';
			ELSIF NOT(MC_BR_SecAddShuttle_1.Execute) THEN
				// Set velocity if the simulation is active
				// If the simulation is active, wiat until the shuttle reached the position
				IF SimActive AND MC_BR_ShReadInfo_Entry.ShuttleInfo.CurrentValues.SegmentPosition.Position >= ENTRY_POSITION_THRESHOLD AND MC_BR_ShReadInfo_Entry.ShuttleInfo.CurrentValues.SegmentPosition.Segment.controlif = Seg_08.controlif(*AND MC_BR_SecReadInfo_SimSector.SectorInfo.ShuttleCount.Count = 0 AND MC_BR_SecReadInfo_SimSector.Valid*) THEN
					MC_BR_SecAddShuttle_1.Velocity	:= ConveyorVelocity;
					MC_BR_SecAddShuttle_1.Execute	:= TRUE;
					EntryState	:= ENTRY_CHECK_TRIGGER;
				ELSIF NOT(SimActive) THEN
					MC_BR_SecAddShuttle_1.Execute	:= TRUE;
					EntryState	:= ENTRY_CHECK_TRIGGER;
				END_IF;
				MC_BR_SecAddShuttle_1.Sector	:= ADR(Sector_2);
				MC_BR_SecAddShuttle_1.Position	:= 0.0;
				MC_BR_SecAddShuttle_1.AdvancedParameters.Mode				:= mcACPTRAK_ADD_CATCH;
				MC_BR_SecAddShuttle_1.AdvancedParameters.VirtualShuttleID	:= VirtShID;
				MC_BR_SecAddShuttle_1.AdvancedParameters.MoveCmd			:= mcACPTRAK_MOV_CMD_ELASTICMOVEVEL;
				MC_BR_SecAddShuttle_1.AdvancedParameters.Velocity			:= ConveyorVelocity;
				MC_BR_SecAddShuttle_1.AdvancedParameters.Acceleration		:= Acceleration;
				MC_BR_SecAddShuttle_1.AdvancedParameters.Deceleration		:= Deceleration;
				MC_BR_SecAddShuttle_1.AdvancedParameters.Direction			:= mcDIR_POSITIVE;
				MC_BR_SecAddShuttle_1.AdvancedParameters.UserID				:= '';
				MC_BR_SecAddShuttle_1.Execute	:= TRUE;
			ELSE
				ErrorInfo	:= 'Error, no SecAddShuttle available';
				State		:= ERROR;
				EntryState	:= ENTRY_ERROR;
			END_IF;

		// Error state, reset all FUBs
		ENTRY_ERROR:
			MC_BR_TrgPointEnable_Entry.Enable		:= FALSE;
			MC_BR_TrgPointReadInfo_Entry.Execute	:= FALSE;
			MC_BR_SecAddShuttle_0.Execute			:= FALSE;
			MC_BR_SecAddShuttle_1.Execute			:= FALSE;
			MC_BR_SecReadInfo_SimSector.Enable		:= FALSE;

			EntryState	:= ENTRY_INIT;
			IF MC_BR_SecAddShuttle_0.Active OR MC_BR_SecAddShuttle_1.Active THEN
				EntryState	:= ENTRY_ABORT_CATCH;
			END_IF;

		// Abort the catch mode
		ENTRY_ABORT_CATCH:
			MC_BR_SecAddShuttle_0.Sector			:= ADR(Sector_2);
			MC_BR_SecAddShuttle_0.AdvancedParameters.Mode	:= mcACPTRAK_ABORT_CATCH;
			MC_BR_SecAddShuttle_0.AdvancedParameters.VirtualShuttleID	:= 0;
			MC_BR_SecAddShuttle_0.Execute			:= TRUE;

			MC_BR_SecAddShuttle_1.Sector			:= ADR(Sector_2);
			MC_BR_SecAddShuttle_1.AdvancedParameters.Mode	:= mcACPTRAK_ABORT_CATCH;
			MC_BR_SecAddShuttle_1.AdvancedParameters.VirtualShuttleID	:= 0;
			MC_BR_SecAddShuttle_1.Execute			:= TRUE;

			IF MC_BR_SecAddShuttle_0.Done AND MC_BR_SecAddShuttle_1.Done THEN
				MC_BR_SecAddShuttle_0.Execute		:= FALSE;
				MC_BR_SecAddShuttle_1.Execute		:= FALSE;
				EntryState	:= ENTRY_INIT;
			ELSIF MC_BR_SecAddShuttle_0.Error OR MC_BR_SecAddShuttle_1.Error THEN
				ErrorInfo	:= 'Error in SecAddShuttle Abort Catch';
				State		:= ERROR;
				EntryState	:= ENTRY_ERROR;
			END_IF;

	END_CASE;

	// Reset the FUB if the station is active and a new shuttle catched
	IF EnableStations THEN
		IF EDGEPOS(MC_BR_SecAddShuttle_0.Active) THEN
			MC_BR_SecAddShuttle_0.Execute		:= FALSE;
			CalcShuttle	:= MC_BR_SecAddShuttle_0.Axis;
		ELSIF MC_BR_SecAddShuttle_0.Error THEN
			ErrorInfo	:= 'Error in SecAddShuttle 0 Entry';
			State		:= ERROR;
			EntryState	:= ENTRY_ERROR;
		END_IF;

		IF EDGEPOS(MC_BR_SecAddShuttle_1.Active) THEN
			MC_BR_SecAddShuttle_1.Execute		:= FALSE;
			CalcShuttle	:= MC_BR_SecAddShuttle_1.Axis;
		ELSIF MC_BR_SecAddShuttle_1.Error THEN
			ErrorInfo	:= 'Error in SecAddShuttle 1 Entry';
			State		:= ERROR;
			EntryState	:= ENTRY_ERROR;
		END_IF;
	END_IF;

	IF MC_BR_SegReadInfo_Entry.Error THEN
		ErrorInfo	:= 'Error in SegReadInfo Entry';
		State		:= ERROR;
		EntryState	:= ENTRY_ERROR;
	END_IF;

	IF MC_BR_SecReadInfo_SimSector.Error THEN
		ErrorInfo	:= 'Error in SecReadInfo SimSector';
		State		:= ERROR;
		EntryState	:= ENTRY_ERROR;
	END_IF;

	// Call the FUBs
	MC_BR_TrgPointEnable_Entry();
	MC_BR_TrgPointReadInfo_Entry();
	MC_BR_ShReadInfo_Entry();

	MC_BR_SecReadInfo_SimSector();
	MC_BR_SegReadInfo_Entry();

END_ACTION
```

#### ExitSegment.st - Exit from the trak to the conveyor
```iecst
(*********************************************************************************
 * Copyright: B&R Industrial Automation GmbH
 * Author:    B&R
 * Created:   July 22, 2025/2:18 PM
 * Description: Exit from the trak to the conveyor, set a cyclic velocity control
 *********************************************************************************)

ACTION ExitSegment:

	// Reset the state machine and all FUBs after a stop or halt command
	// Avoid shuttles to go on the conveyor
	IF (Paused OR EnableStations = FALSE) AND ExitState <> EXIT_INIT THEN
		ExitState	:= EXIT_ERROR;
	END_IF;

	CASE ExitState OF
		// Wait for enable the station
		EXIT_INIT:
			IF EnableStations AND NOT(Paused) THEN
				AddTicket	:= TRUE; // Allow one shuttle through barrier
				ExitState	:= EXIT_CHECK_TRIGGER;
				MC_BR_BarrierReadInfo_Exit.Enable	:= TRUE;
			END_IF;

		// Check for a shuttle passing the trigger
		EXIT_CHECK_TRIGGER:
			MC_BR_TrgPointEnable_Exit.Enable		:= TRUE;

			// If the barrier is still closed, add another ticket
			IF MC_BR_BarrierReadInfo_Exit.BarrierInfo.Status = mcACPTRAK_BARRIER_CLOSED THEN
				AddTicket	:= TRUE; // Allow one shuttle through barrier
			END_IF;

			IF MC_BR_TrgPointEnable_Exit.Valid AND MC_BR_TrgPointEnable_Exit.EventCount > 0 THEN
				ExitState	:= EXIT_GET_SHUTTLE;
			ELSIF MC_BR_TrgPointEnable_Exit.Error THEN
				ErrorInfo	:= 'Error in TrgPointEnable Exit';
				State		:= ERROR;
				ExitState	:= EXIT_ERROR;
			END_IF;

		// Get the shuttle exiting the trak
		EXIT_GET_SHUTTLE:
			MC_BR_TrgPointReadInfo_Exit.Execute	:= TRUE;

			IF MC_BR_TrgPointReadInfo_Exit.Done THEN
				MC_BR_TrgPointReadInfo_Exit.Execute	:= FALSE;
				ExitShuttle	:= MC_BR_TrgPointReadInfo_Exit.TrgPointInfo.Axis;
				ExitState		:= EXIT_GET_SHUTTLEID;
			ELSIF MC_BR_TrgPointReadInfo_Exit.Error THEN
				ErrorInfo	:= 'Error in TrgPointReadInfo Exit';
				State		:= ERROR;
				ExitState	:= EXIT_ERROR;
			END_IF;

		// Read shuttle information
		EXIT_GET_SHUTTLEID:
			MC_BR_ShReadInfo_Exit.Axis		:= ADR(ExitShuttle);
			MC_BR_ShReadInfo_Exit.Enable	:= TRUE;

			IF MC_BR_ShReadInfo_Exit.Valid THEN
				MC_BR_ShReadInfo_Exit.Enable	:= FALSE;
				ExitState	:= EXIT_CYCMOVEVEL;

				Message		:= 'Shuttle "';
				brsstrcat(ADR(Message),ADR(MC_BR_ShReadInfo_Exit.ShuttleInfo.AdditionalInfo.UserID));
				brsstrcat(ADR(Message),ADR('" left the trak and entered the conveyor'));
				AddMessage	:= TRUE;
				AddImage	:= 1;
			ELSIF MC_BR_ShReadInfo_Exit.Error THEN
				ErrorInfo	:= 'Error in ShReadInfo Exit';
				State		:= ERROR;
				ExitState	:= EXIT_ERROR;
			END_IF;

		// Set a cyclic MoveVel to the shuttle with the same speed as the conveyor
		EXIT_CYCMOVEVEL:
			FOR Index := 0 TO MAX_SHUTTLES_MIN_ONE DO
				IF Shuttle[Index].controlif	= ExitShuttle.controlif AND State = READY THEN
					MC_BR_MoveCyclicTcpVel_0[Index].Enable	:= TRUE;
					EXIT;
				END_IF;
			END_FOR;
			IF MC_BR_MoveCyclicTcpVel_0[Index].Valid THEN
				ExitState	:= EXIT_CHECK_TRIGGER;
			END_IF;

		// Error state, reset all FUBs
		EXIT_ERROR:
			MC_BR_TrgPointEnable_Exit.Enable	:= FALSE;
			MC_BR_TrgPointReadInfo_Exit.Execute	:= FALSE;

			MC_BR_ShReadInfo_Exit.Enable		:= FALSE;

			MC_BR_BarrierCmd_Exit.Execute		:= FALSE;

			MC_BR_TrgPointEnable_CheckFree.Enable	:= FALSE;

			ExitState	:= EXIT_INIT;

	END_CASE;

	MC_BR_TrgPointEnable_CheckFree.Enable		:= ExitState <> EXIT_ERROR AND ExitState <> EXIT_INIT;
	IF MC_BR_TrgPointEnable_CheckFree.Valid AND MC_BR_TrgPointEnable_CheckFree.EventCount > 0 THEN
		MC_BR_TrgPointEnable_CheckFree.Enable	:= FALSE;
		AddTicket	:= TRUE;
	ELSIF MC_BR_TrgPointEnable_CheckFree.Error THEN
		ErrorInfo	:= 'Error in TrgPointEnable CheckFree';
		State		:= ERROR;
		ExitState	:= EXIT_ERROR;
	END_IF;

	// If no movement of the conveyor is active, close the barrier to prevent shuttles going onto the conveyor
	// Additionally close the barrier during the cleaning phase of the conveyor
	IF (MpAxisBasic_0.MoveActive = FALSE OR StopConveyor OR Paused OR (State >= CLEAN_CONVEYOR AND State <= CLEAN_CONVEYOR_ABORT)) AND
		MC_BR_BarrierReadInfo_Exit.BarrierInfo.Status <> mcACPTRAK_BARRIER_CLOSED AND MC_BR_BarrierReadInfo_Exit.Valid THEN

		AddTicket	:= FALSE;
		MC_BR_BarrierCmd_Exit.Command	:= mcACPTRAK_BARRIER_CLOSE;
		MC_BR_BarrierCmd_Exit.Execute	:= TRUE;

	// Open the conveyor when the movement is active
	ELSIF MpAxisBasic_0.MoveActive AND StopConveyor = FALSE AND Paused = FALSE AND AddTicket AND MC_BR_BarrierReadInfo_Exit.BarrierInfo.RemainingTickets = 0 AND
		(MC_BR_BarrierReadInfo_Exit.BarrierInfo.Status = mcACPTRAK_BARRIER_CLOSED OR MC_BR_BarrierReadInfo_Exit.BarrierInfo.Status = mcACPTRAK_BARRIER_TICKETING) AND MC_BR_BarrierReadInfo_Exit.Valid THEN

		AddTicket	:= FALSE;
		MC_BR_BarrierCmd_Exit.AdvancedParameters.TicketCount	:= 1;
		MC_BR_BarrierCmd_Exit.Command	:= mcACPTRAK_BARRIER_ADD_TICKETS;
		MC_BR_BarrierCmd_Exit.Execute	:= TRUE;
	END_IF;

	// Reset the barrier command
	IF MC_BR_BarrierCmd_Exit.Done THEN
		MC_BR_BarrierCmd_Exit.Execute	:= FALSE;
	ELSIF MC_BR_BarrierCmd_Exit.Error THEN
		ErrorInfo	:= 'Error in BarrierCmd Exit';
		State		:= ERROR;
		ExitState	:= EXIT_ERROR;
	END_IF;

	// Check error for reading barrier info
	IF MC_BR_BarrierReadInfo_Exit.Error THEN
		MC_BR_BarrierReadInfo_Exit.Enable	:= FALSE;
		ErrorInfo	:= 'Error in BarrierReadInfo Exit';
		State		:= ERROR;
		ExitState	:= EXIT_ERROR;
	END_IF;

	// Call the FUBs
	MC_BR_TrgPointEnable_Exit();
	MC_BR_TrgPointReadInfo_Exit();

	MC_BR_ShReadInfo_Exit();

	MC_BR_BarrierCmd_Exit();
	MC_BR_BarrierReadInfo_Exit();

	MC_BR_TrgPointEnable_CheckFree();

END_ACTION
```

#### Clear.st - Clear station
```iecst
(*********************************************************************************
 * Copyright: B&R Industrial Automation GmbH
 * Author:    B&R
 * Created:   July 22, 2025/2:18 PM
 * Description: Clear station to move the shuttles elastic after the conveyor
 *********************************************************************************)

ACTION Clear:

	// Reset the state machine and all FUBs after a stop command
	IF EnableStations = FALSE AND ClearState <> CLEAR_INIT THEN
		ClearState	:= CLEAR_ERROR;
	END_IF;

	// Reset the state machine after a Halt command
	IF Paused THEN
		ClearState	:= CLEAR_ERROR;
	END_IF;

	CASE ClearState OF
		// Wait for enabling the station
		CLEAR_INIT:
			IF EnableStations THEN
				ClearState	:= CLEAR_CHECK_TRIGGER;
			END_IF;

		// Check for trigger event
		CLEAR_CHECK_TRIGGER:
			MC_BR_TrgPointEnable_Clear.Enable		:= TRUE;

			IF MC_BR_TrgPointEnable_Clear.Valid AND MC_BR_TrgPointEnable_Clear.EventCount > 0 THEN
				ClearState	:= CLEAR_GET_SHUTTLE;
			ELSIF MC_BR_TrgPointEnable_Clear.Error THEN
				ErrorInfo	:= 'Error in TrgPointEnable Clear';
				State		:= ERROR;
				ClearState	:= CLEAR_ERROR;
			END_IF;

		// Get the passed shuttle
		CLEAR_GET_SHUTTLE:
			MC_BR_TrgPointReadInfo_Clear.Execute	:= TRUE;

			IF MC_BR_TrgPointReadInfo_Clear.Done THEN
				MC_BR_TrgPointReadInfo_Clear.Execute	:= FALSE;
				ClearShuttle	:= MC_BR_TrgPointReadInfo_Clear.TrgPointInfo.Axis;
				ClearState		:= CLEAR_MOVE_SH_ELASTIC;
			ELSIF MC_BR_TrgPointReadInfo_Clear.Error THEN
				ErrorInfo	:= 'Error in TrgPointReadInfo Clear';
				State		:= ERROR;
				ClearState	:= CLEAR_ERROR;
			END_IF;

		// Move the shuttle elastic
		CLEAR_MOVE_SH_ELASTIC:
			MC_BR_ElasticMoveVel_Clear.Axis			:= ADR(ClearShuttle);
			MC_BR_ElasticMoveVel_Clear.Velocity		:= Velocity;
			MC_BR_ElasticMoveVel_Clear.Acceleration	:= Acceleration;
			MC_BR_ElasticMoveVel_Clear.Deceleration	:= Deceleration;
			MC_BR_ElasticMoveVel_Clear.Direction	:= mcDIR_POSITIVE;
			MC_BR_ElasticMoveVel_Clear.Execute		:= NOT(Paused);

			// If a global stop command is executed, reset the command and go back to the trigger state
			IF EDGEPOS(MC_BR_ElasticMoveVel_Clear.Active) OR (MC_BR_ElasticMoveVel_Clear.Error AND MC_BR_AsmStop_0.Execute) THEN
				MC_BR_ElasticMoveVel_Clear.Execute	:= FALSE;
				ClearState	:= CLEAR_CHECK_TRIGGER;
			ELSIF MC_BR_ElasticMoveVel_Clear.Error THEN
				ErrorInfo	:= 'Error in ElasticMoveVel Clear';
				State		:= ERROR;
				ClearState	:= CLEAR_ERROR;
			END_IF;

		// Error state, reset all FUBs
		CLEAR_ERROR:
			MC_BR_TrgPointEnable_Clear.Enable		:= FALSE;
			MC_BR_TrgPointReadInfo_Clear.Execute	:= FALSE;
			MC_BR_ElasticMoveVel_Clear.Execute		:= FALSE;

			ClearState	:= CLEAR_INIT;

	END_CASE;

	// Call the FUBs
	MC_BR_TrgPointEnable_Clear();
	MC_BR_TrgPointReadInfo_Clear();
	MC_BR_ElasticMoveVel_Clear();

END_ACTION
```

#### AddNewShuttle.st - Station to add a new shuttle
```iecst
(*********************************************************************************
 * Copyright: B&R Industrial Automation GmbH
 * Author:    B&R
 * Created:   July 22, 2025/2:18 PM
 * Description: Add a new shuttle to the trak if possible
 *********************************************************************************)

ACTION AddNewShuttle:

	// Reset the state machine and all FUBs after a stop command
	IF OpenBarrier OR EDGENEG(EnableStations) THEN
		AddShuttleState	:= ADDSHUTTLE_RESET;
	END_IF;

	CASE AddShuttleState OF
		// Wait for enabling the station
		ADDSHUTTLE_INIT:
			IF AddShuttle AND EnableStations AND MC_BR_AsmReadInfo_0.AssemblyInfo.ShuttleCount.Count <= MAX_SHUTTLES THEN
				AddShuttleState	:= ADDSHUTTLE_CLOSE_BARRIER;
			END_IF;

		// Close the barrier to avoid a shuttle to be created on another one
		ADDSHUTTLE_CLOSE_BARRIER:
			MC_BR_SecReadInfo_AddShuttle.Enable			:= TRUE;

			MC_BR_BarrierCmd_AddShuttle.Command			:= mcACPTRAK_BARRIER_CLOSE;
			MC_BR_BarrierCmd_AddShuttle.Execute			:= TRUE;

			IF MC_BR_BarrierCmd_AddShuttle.Done THEN
				MC_BR_BarrierCmd_AddShuttle.Execute		:= FALSE;
				// Simulation: immediate add | Hardware: power cycle segment first
				IF SimActive THEN
					AddShuttleState	:= ADDSHUTTLE_ADD_SHUTTLE;
				ELSE
					BarrierClosed_AddShuttle	:= TRUE; // Signal UI that user can place shuttle
					AddShuttleState	:= ADDSHUTTLE_POWER_OFF_SEGMENT;
				END_IF;
			ELSIF MC_BR_BarrierCmd_AddShuttle.Error THEN
				ErrorInfo		:= 'Error in BarrierCmd AddShuttle';
				State			:= ERROR;
				AddShuttleState	:= ADDSHUTTLE_ERROR;
			END_IF;

		// Add a shuttle to the trak
		ADDSHUTTLE_ADD_SHUTTLE:
			MC_BR_SecAddShuttle_AddShuttle.Sector		:= ADR(Sector_1);
			MC_BR_SecAddShuttle_AddShuttle.Position		:= AddPosition;
			MC_BR_SecAddShuttle_AddShuttle.Velocity		:= Velocity;
			MC_BR_SecAddShuttle_AddShuttle.AdvancedParameters.Mode			:= mcACPTRAK_ADD_IMMEDIATE;
			MC_BR_SecAddShuttle_AddShuttle.AdvancedParameters.MoveCmd		:= mcACPTRAK_MOV_CMD_ELASTICMOVEVEL;
			MC_BR_SecAddShuttle_AddShuttle.AdvancedParameters.Direction		:= mcDIR_POSITIVE;
			MC_BR_SecAddShuttle_AddShuttle.AdvancedParameters.Velocity		:= Velocity;
			MC_BR_SecAddShuttle_AddShuttle.AdvancedParameters.Acceleration	:= Acceleration;
			MC_BR_SecAddShuttle_AddShuttle.AdvancedParameters.Deceleration	:= Deceleration;
			MC_BR_SecAddShuttle_AddShuttle.AdvancedParameters.UserID		:= UserID;
			// Only add shuttle when sector is at rest, data is valid, and no other shuttles present
			IF MC_BR_SecReadInfo_AddShuttle.SectorInfo.InRest AND MC_BR_SecReadInfo_AddShuttle.Valid AND MC_BR_SecReadInfo_AddShuttle.SectorInfo.ShuttleCount.Count = 0 THEN
				MC_BR_SecAddShuttle_AddShuttle.Execute	:= TRUE;
				AddShuttleState	:= ADDSHUTTLE_CHECK_CREATED;
			END_IF;

		// Check for shuttle created
		ADDSHUTTLE_CHECK_CREATED:
			IF MC_BR_SecAddShuttle_AddShuttle.Axis.controlif <> AxisOld.controlif THEN
				MC_BR_SecAddShuttle_AddShuttle.Execute	:= FALSE;
				AddShuttleState	:= ADDSHUTTLE_OPEN_BARRIER;
			ELSIF MC_BR_SecAddShuttle_AddShuttle.Error THEN
				ErrorInfo	:= 'Error in SecAddShuttle AddShuttle';
				State		:= ERROR;
				AddShuttleState	:= ADDSHUTTLE_ERROR;
			END_IF;
			// Check if new shuttle created
			AxisOld	:= MC_BR_SecAddShuttle_AddShuttle.Axis; // Store reference to detect controlif change (new shuttle created)

		// Power off the segment
		ADDSHUTTLE_POWER_OFF_SEGMENT:
			MC_BR_SegPowerOff_AddShuttle.Segment		:= ADR(Seg_01);
			IF MC_BR_SecReadInfo_AddShuttle.SectorInfo.InRest AND MC_BR_SecReadInfo_AddShuttle.Valid THEN
				MC_BR_SegPowerOff_AddShuttle.Execute	:= TRUE;
			END_IF;

			IF MC_BR_SegPowerOff_AddShuttle.Done THEN
				MC_BR_SegPowerOff_AddShuttle.Execute	:= FALSE;
				AddShuttleState	:= ADDSHUTTLE_POWER_ON_SEGMENT;
			ELSIF MC_BR_SegPowerOff_AddShuttle.Error THEN
				ErrorInfo		:= 'Error in SegPowerOff AddShuttle';
				State			:= ERROR;
				AddShuttleState	:= ADDSHUTTLE_ERROR;
			END_IF;

		// Power on the segment
		ADDSHUTTLE_POWER_ON_SEGMENT:
			MC_BR_SegPowerOn_AddShuttle.Segment		:= ADR(Seg_01);
			MC_BR_SegPowerOn_AddShuttle.Execute		:= ConfirmShuttleAdded;

			IF MC_BR_SegPowerOn_AddShuttle.Done THEN
				MC_BR_SegPowerOn_AddShuttle.Execute	:= FALSE;
				AddShuttleState	:= ADDSHUTTLE_GET_SHUTTLE;
			ELSIF MC_BR_SegPowerOn_AddShuttle.Error THEN
				ErrorInfo		:= 'Error in SegPowerOn AddShuttle';
				State			:= ERROR;
				AddShuttleState	:= ADDSHUTTLE_ERROR;
			END_IF;

		// Get shuttle reference for real hardware
		ADDSHUTTLE_GET_SHUTTLE:
			MC_BR_SecGetShuttle_AddShuttle.Sector		:= ADR(Sector_3);
			MC_BR_SecGetShuttle_AddShuttle.Enable		:= TRUE;

			IF MC_BR_SecGetShuttle_AddShuttle.Valid THEN
				MC_BR_SecGetShuttle_AddShuttle.Next		:= FALSE;
				// If Continue is pressed check how many shuttles are on the trak
				// If no shuttles are on the trak open the barrier, if at least one is, set the UserID
				IF MC_BR_SecGetShuttle_AddShuttle.TotalCount > 0 THEN
					AddedShuttle	:= MC_BR_SecGetShuttle_AddShuttle.Axis;
					AddShuttleState	:= ADDSHUTTLE_SET_USERID;
				ELSE
					MC_BR_SecGetShuttle_AddShuttle.Enable	:= FALSE;
					AddShuttleState	:= ADDSHUTTLE_OPEN_BARRIER;
				END_IF;
			ELSIF MC_BR_SecGetShuttle_AddShuttle.Error THEN
				ErrorInfo		:= 'Error in SecGetShuttle AddShuttle';
				State			:= ERROR;
				AddShuttleState	:= ADDSHUTTLE_ERROR;
			END_IF;

		// Set the UserID for the shuttle
		ADDSHUTTLE_SET_USERID:
			MC_BR_ShSetUserID_AddShuttle.Axis			:= ADR(AddedShuttle);
			MC_BR_ShSetUserID_AddShuttle.UserID			:= UserID;
			MC_BR_ShSetUserID_AddShuttle.Execute		:= TRUE;

			IF MC_BR_ShSetUserID_AddShuttle.Done THEN
				MC_BR_ShSetUserID_AddShuttle.Execute	:= FALSE;
				AddShuttleState	:= ADDSHUTTLE_MOVESHUTTLE;
			ELSIF MC_BR_ShSetUserID_AddShuttle.Error THEN
				ErrorInfo		:= 'Error in ShSetUserID AddShuttle';
				State			:= ERROR;
				AddShuttleState	:= ADDSHUTTLE_ERROR;
			END_IF;

		// Start a movement for the shuttle
		ADDSHUTTLE_MOVESHUTTLE:
			MC_BR_ElasticMoveVel_AddShuttle.Axis		:= ADR(AddedShuttle);
			MC_BR_ElasticMoveVel_AddShuttle.Direction	:= mcDIR_POSITIVE;
			MC_BR_ElasticMoveVel_AddShuttle.Velocity	:= Velocity;
			MC_BR_ElasticMoveVel_AddShuttle.Acceleration:= Acceleration;
			MC_BR_ElasticMoveVel_AddShuttle.Deceleration:= Deceleration;
			MC_BR_ElasticMoveVel_AddShuttle.Execute		:= TRUE;

			IF EDGEPOS(MC_BR_ElasticMoveVel_AddShuttle.Active) THEN
				MC_BR_ElasticMoveVel_AddShuttle.Execute	:= FALSE;

				// If all shuttles are read, power on the segment
				IF MC_BR_SecGetShuttle_AddShuttle.RemainingCount = 0 THEN
					MC_BR_SecGetShuttle_AddShuttle.Enable	:= FALSE;
					AddShuttleState	:= ADDSHUTTLE_OPEN_BARRIER;
				ELSE
					MC_BR_SecGetShuttle_AddShuttle.Next	:= TRUE;
					AddShuttleState	:= ADDSHUTTLE_GET_SHUTTLE;
				END_IF;
			ELSIF MC_BR_ElasticMoveVel_AddShuttle.Error THEN
				ErrorInfo		:= 'Error in ElasticMoveVel AddShuttle';
				State			:= ERROR;
				AddShuttleState	:= ADDSHUTTLE_ERROR;
			ELSIF MC_BR_SecGetShuttle_AddShuttle.Error THEN
				ErrorInfo		:= 'Error in SecGetShuttle AddShuttle';
				State			:= ERROR;
				AddShuttleState	:= ADDSHUTTLE_ERROR;
			END_IF;

		// Open the barrier again
		ADDSHUTTLE_OPEN_BARRIER:
			MC_BR_BarrierCmd_AddShuttle.Command			:= mcACPTRAK_BARRIER_OPEN;
			MC_BR_BarrierCmd_AddShuttle.Execute			:= TRUE;

			IF MC_BR_BarrierCmd_AddShuttle.Done THEN
				MC_BR_BarrierCmd_AddShuttle.Execute		:= FALSE;
				AddShuttle					:= FALSE;
				ConfirmShuttleAdded			:= FALSE;
				BarrierClosed_AddShuttle	:= FALSE;
				AddShuttleState	:= ADDSHUTTLE_INIT;
			ELSIF MC_BR_BarrierCmd_AddShuttle.Error THEN
				ErrorInfo		:= 'Error in BarrierCmd AddShuttle';
				State			:= ERROR;
				AddShuttleState	:= ADDSHUTTLE_ERROR;
			END_IF;

		// Reset the station and open the barrier
		ADDSHUTTLE_RESET:
			MC_BR_BarrierCmd_AddShuttle.Execute			:= FALSE;
			OpenBarrier			:= FALSE;
			AddShuttleState		:= ADDSHUTTLE_OPEN_BARRIER;

		// Error state, reset all FUBs
		ADDSHUTTLE_ERROR:
			MC_BR_SecAddShuttle_AddShuttle.Execute		:= FALSE;
			MC_BR_SecReadInfo_AddShuttle.Enable			:= FALSE;
			MC_BR_BarrierCmd_AddShuttle.Execute			:= FALSE;

			AddShuttleState		:= ADDSHUTTLE_INIT;

	END_CASE;

	IF MC_BR_SecReadInfo_AddShuttle.Error THEN
		MC_BR_SecReadInfo_AddShuttle.Enable			:= FALSE;
		ErrorInfo		:= 'Error in SecReadInfo AddShuttle';
		State			:= ERROR;
		AddShuttleState	:= ADDSHUTTLE_ERROR;
	END_IF;

	// Call the FUBs
	MC_BR_SecAddShuttle_AddShuttle();
	MC_BR_SecReadInfo_AddShuttle();
	MC_BR_BarrierCmd_AddShuttle();

	MC_BR_SegPowerOff_AddShuttle();
	MC_BR_SegPowerOn_AddShuttle();
	MC_BR_SecGetShuttle_AddShuttle();
	MC_BR_ShSetUserID_AddShuttle();
	MC_BR_ElasticMoveVel_AddShuttle();

END_ACTION
```

#### CalcAutomaticVelocity.st - Calculate automatic velocity adjustment
```iecst
(*********************************************************************************
 * Copyright: B&R Industrial Automation GmbH
 * Author:    B&R
 * Created:   July 24, 2025/10:46 AM
 * Description: Calculate the automatic velocity adjustment
 *********************************************************************************)

ACTION CalcAutomaticVelocity:

	MC_BR_ShReadInfo_Calc.Axis			:= ADR(CalcShuttle);
	MC_BR_ShReadInfo_Calc.Enable		:= AutomaticVelocityAdjustment AND CalcShuttle.controlif <> 0 AND EnableStations;

	// Restart the FUB when a new shuttle is available
	IF CalcShuttle.controlif <> OldShuttle_Calc.controlif THEN
		MC_BR_ShReadInfo_Calc.Enable	:= FALSE;
	END_IF;

	OldShuttle_Calc	:= CalcShuttle;

	IF MC_BR_ShReadInfo_Calc.Error THEN
		ErrorInfo	:= 'Error in ShReadInfo Calc';
		State		:= ERROR;
	END_IF;

	// Call the FUBs
	MC_BR_ShReadInfo_Calc();

	// Get the velocity if the shuttle is real and on the first segment after the conveyor
	IF MC_BR_ShReadInfo_Calc.Valid AND MC_BR_ShReadInfo_Calc.ShuttleInfo.CurrentValues.SegmentPosition.Segment.controlif = Seg_08.controlif AND
		MC_BR_ShReadInfo_Calc.ShuttleInfo.CurrentValues.SegmentPosition.Position < CLEAR_POSITION_THRESHOLD AND NOT(MC_BR_ShReadInfo_Calc.ShuttleInfo.AdditionalInfo.Virtual) AND
		MC_BR_ShReadInfo_Calc.ShuttleInfo.CurrentValues.Velocity <> 0 THEN
		ConveyorVelocity	:= MC_BR_ShReadInfo_Calc.ShuttleInfo.CurrentValues.Velocity;
	// If the shuttle left the segment, but no other shuttle is available, set the maximum speed
	ELSIF MC_BR_ShReadInfo_Calc.Valid AND NOT(MC_BR_ShReadInfo_Calc.ShuttleInfo.AdditionalInfo.Virtual) THEN
		ConveyorVelocity	:= 2.0; // Fallback to maximum speed when no shuttle detected
	END_IF;

END_ACTION
```

- Visualisation Logical/mappView (not shown)

### Package Logical/Scene - Scene files

- gAssembly_1.wsp (not shown)

- mappView.bat - Script to open the mappView visu in Chrome (not shown)

Listed in the project but not available here: Logical/Global.typ, Logical/Global.var
